// TIA Portal V19 program export: 1 tag tables, 0 data types, 19 data blocks, 18 code blocks (in call order from the OBs), 296 instance data blocks

VAR_GLOBAL   // PLC tag table "Default tag table"
   "CPU RUN" AT %I0.0 : Bool;
   "SPARE(1)" AT %I0.1 : Bool;
   "SPARE(2)" AT %I0.2 : Bool;
   "P-201 A RO 1 FEED PUMP TRIP" AT %I0.3 : Bool;
   "P-201 B RO 1 FEED PUMP TRIP" AT %I0.4 : Bool;
   "P-201 C RO 1 FEED PUMP TRIP" AT %I0.5 : Bool;
   "P-301 A RO 1 HPP PUMP TRIP" AT %I0.6 : Bool;
   "P-301 B RO B HPP PUMP TRIP" AT %I0.7 : Bool;
   "P-401 A RO 2 FEED PUMP TRIP" AT %I1.0 : Bool;
   "P-401 B RO 2 FEED PUMP TRIP" AT %I1.1 : Bool;
   "P-401 C RO 2 FEED PUMP TRIP" AT %I1.2 : Bool;
   "P 401 A RO 2 HPP PUMP TRIP" AT %I1.3 : Bool;
   "P-401 B RO 2 HPP PUMP TRIP" AT %I1.4 : Bool;
   "LPS 301 RO 1" AT %I1.5 : Bool;
   "P-202 A RO 1 FEED PUMP" AT %Q0.0 : Bool;
   "P-202 B RO 1 FEED PUMP" AT %Q0.1 : Bool;
   "P-202 C RO 1 FEED PUMP" AT %Q0.2 : Bool;
   "P-301 A RO 1 HPP PUMP" AT %Q0.3 : Bool;
   "P-301 B RO 1 HPP PUMP" AT %Q0.4 : Bool;
   "P-401 A RO 2 FEED PUMP" AT %Q0.5 : Bool;
   "P-401 B RO 2 FEED PUMP" AT %Q0.6 : Bool;
   "P-401 C RO 2 FEED PUMP" AT %Q0.7 : Bool;
   "P-402  A RO 2 HPP" AT %Q1.0 : Bool;
   "P-402 B" AT %Q1.1 : Bool;
   "HPS-301 RO 1 PRESSURE SWITCH" AT %I8.0 : Bool;
   "LPS-302 RO 1 PRESSURE SWITCH" AT %I8.1 : Bool;
   "HPS-302 RO 1 PRESSURE SWITCH" AT %I8.2 : Bool;
   "LPS-401 RO 2 PRESSURE SWITCH" AT %I8.3 : Bool;
   "HPS-401 RO 2 PRESSURE SWITCH" AT %I8.4 : Bool;
   "LPS-402 RO 2 PRESSURE SWITCH" AT %I8.5 : Bool;
   "HPS-402 RO 2 PRESSURE SWITCH" AT %I8.6 : Bool;
   "DP-703 RO 1 DOSER LEVEL SWITCH" AT %I8.7 : Bool;
   "DP-704 RO 1 DOSER LEVEL SWITCH" AT %I9.0 : Bool;
   "DP-705 RO 1 DOSER LEVEL SWITCH" AT %I9.1 : Bool;
   "P-501 A EDI FEED PUMP TRIP" AT %I9.2 : Bool;
   "P-501 B EDI FEED PUMP TRIP" AT %I9.3 : Bool;
   "P-501 C EDI FEED PUMP TRIP" AT %I9.4 : Bool;
   "EDI 501 A TRIP" AT %I9.5 : Bool;
   "EDI 501 B TRIP" AT %I9.6 : Bool;
   "P-501 A EDI FEED PUMP" AT %Q8.0 : Bool;
   "P-501 B EDI FEED PUMP" AT %Q8.1 : Bool;
   "P-501 C EDI FEED PUMP" AT %Q8.2 : Bool;
   "EDI 501" AT %Q8.3 : Bool;
   "EDI 502" AT %Q8.4 : Bool;
   "DP 703" AT %Q8.5 : Bool;
   "DP 704" AT %Q8.6 : Bool;
   "DP 705" AT %Q8.7 : Bool;
   "ABV 301" AT %Q9.0 : Bool;
   "ABV 302" AT %Q9.1 : Bool;
   "AGLV-301" AT %Q9.2 : Bool;
   "AGLV-302" AT %Q9.3 : Bool;
   "AGLV-401" AT %Q9.4 : Bool;
   "AGLV-402" AT %Q9.5 : Bool;
   "AGLV-501" AT %Q9.6 : Bool;
   "AGLV-502" AT %Q9.7 : Bool;
   "P-201 A RO 1 FEED PUMP FEED BACK" AT %I12.0 : Bool;
   "P-201 B RO 1 FEED PUMP FEED BACK" AT %I12.1 : Bool;
   "P-201 C RO 1 FEED PUMP FEED BACK" AT %I12.2 : Bool;
   "P-301 A RO 1 HPP PUMP FEED BACK" AT %I12.3 : Bool;
   "P-301 B RO 1 HPP PUMP FEED BACK" AT %I12.4 : Bool;
   "P-401 A R0 2 FEED PUMP FEED BACK" AT %I12.5 : Bool;
   "P-401 B RO 2 FEED PUMP FEED BACK" AT %I12.6 : Bool;
   "P-401 C RO 2 FEED PUMP FEED BACK" AT %I12.7 : Bool;
   "P-402 A RO 2 HPP PUMP FEED BACK" AT %I13.0 : Bool;
   "P-402 B RO 2 HPP PUMP FEED BACK" AT %I13.1 : Bool;
   "P-501 A EDI FEED PUMP FEED BACK" AT %I13.2 : Bool;
   "P-501 B EDI FEED PUMP FEED BACK" AT %I13.3 : Bool;
   "P-501 C EDI FEED PUMP FEED BACK" AT %I13.4 : Bool;
   "SPARE(3)" AT %I13.5 : Bool;
   "ABFV-301 FEED BACK OPEN" AT %I13.6 : Bool;
   "ABFV-301 FEED BACK CLOSE" AT %I13.7 : Bool;
   "ABFV-302 OPEN FEED BACK" AT %I16.0 : Bool;
   "ABFV-302 CLOSE FEED BACK" AT %I16.1 : Bool;
   "AGLV-301 OPEN FEED BACK" AT %I16.2 : Bool;
   "AGLV-301 CLOSE FEED BACK" AT %I16.3 : Bool;
   "AGLV-302 OPEN FEED BACK" AT %I16.4 : Bool;
   "AGLV-302 CLOSE FEED BACK" AT %I16.5 : Bool;
   "AGLV-401 OPEN FEED BACK" AT %I16.6 : Bool;
   "AGLV-401 CLOSE FEED BACK" AT %I16.7 : Bool;
   "AGLV-402 OPEN FEED BACK" AT %I17.0 : Bool;
   "AGLV-402 CLOSE FEED BACK" AT %I17.1 : Bool;
   "AGLV-501OPEN FEED BACK" AT %I17.2 : Bool;
   "AGLV-501 CLOSE FEED BACK" AT %I17.3 : Bool;
   "AGLV-502 OPEN FEED BACK" AT %I17.4 : Bool;
   "AGLV-502 CLOSE FEED BACK" AT %I17.5 : Bool;
   "SPARE(4)" AT %I17.6 : Bool;
   "SPARE(5)" AT %I17.7 : Bool;
   "OXIDATION REDUCTION POTENTIO METER 301" AT %IW144 : Int;
   "CONDUCTIVITY INDUCTOR CUM TRANSMITTER 301" AT %IW146 : Int;
   "PH INDICATOR CUM TRANSMITTER 301" AT %IW148 : Int;
   "PH INDICATOR CUM TRANSMITTER 302" AT %IW150 : Int;
   "CONDUCTIVITY INDICATOR CUM TRANSMITTER 302" AT %IW152 : Int;
   "LEVEL TRANSMITTER 401" AT %IW154 : Int;
   "PH INDICATOR CUM TRANSMITTER 401" AT %IW156 : Int;
   "CONDUCTIVITY INDICATOR CUM TRANSMITTER 401" AT %IW158 : Int;
   "CONFUCTIVITY INDICATOR CUM TRANSMITTER 402" AT %IW160 : Int;
   "PH INDICATOR CUM TRANSMITTER 402" AT %IW162 : Int;
   "LEVEL TRANSMITTER 501" AT %IW164 : Int;
   "FLOW INDICATOR TOTALOZER 501" AT %IW166 : Int;
   "PRESSURE TRANSMITTER 501" AT %IW168 : Int;
   "FLOW INDICATOR TRANSMITTER 502" AT %IW170 : Int;
   "PRESSURE TRANSMITTER 502" AT %IW172 : Int;
   "PRESSURE TRANSMITTER 503" AT %IW174 : Int;
   "PRESSURE TRANSMITTER 504" AT %IW176 : Int;
   "PRESSURE TRANSMITTER 505" AT %IW178 : Int;
   "PRESSURE TRANSMITTER 506" AT %IW180 : Int;
   "PH INDICATOR CUM TRANSMITTER 501" AT %IW182 : Int;
   "PH INDICATOR CUM TRANSMITTER 502" AT %IW184 : Int;
   "RESISTIVITY CUM TRANSMITTER 501" AT %IW186 : Int;
   "RESISTIVITY CUM TRANSMITTER 502" AT %IW188 : Int;
   "LEVEL TRANSMITTER 502" AT %IW190 : Int;
   "FLOW INDICATOR TRANSMITTER 503" AT %IW192 : Int;
   "FLOW INDICATOR TRANSMITTER 504" AT %IW194 : Int;
   "FLOW INDICATOR TRANSMITTER 505" AT %IW196 : Int;
   "FLOW INDICATOR TRANSMITTER 506" AT %IW198 : Int;
   "FLOW INDICATOR TRANSMITTER 507" AT %IW200 : Int;
   "FLOW INDICATOR TRANSMITTER 508" AT %IW202 : Int;
   "SPARE(6)" AT %IW204 : Int;
   "SPARE(7)" AT %IW206 : Int;
   "SPARE(8)" AT %I9.7 : Bool;
   Tag_1 AT %Q1.2 : Bool;
   Tag_2 AT %I1.6 : Bool;
   Clock_Byte AT %MB0 : Byte;
   Clock_10Hz AT %M0.0 : Bool;
   Clock_5Hz AT %M0.1 : Bool;
   "Clock_2.5Hz" AT %M0.2 : Bool;
   Clock_2Hz AT %M0.3 : Bool;
   "Clock_1.25Hz" AT %M0.4 : Bool;
   Clock_1Hz AT %M0.5 : Bool;
   "Clock_0.625Hz" AT %M0.6 : Bool;
   "Clock_0.5Hz" AT %M0.7 : Bool;
   System_Byte AT %MB1 : Byte;
   FirstScan AT %M1.0 : Bool;
   DiagStatusUpdate AT %M1.1 : Bool;
   AlwaysTRUE AT %M1.2 : Bool;
   AlwaysFALSE AT %M1.3 : Bool;
   "PLC_2 HOOTER" AT %M2.0 : Bool;
   "SET TIME" AT %MW4 : Int;
   "LT 201" AT %MD6 : Real;
   TAG122 AT %M2.1 : Bool;
   TEST_1 AT %M2.2 : Bool;
   TEST_2 AT %M2.3 : Bool;
   TEST_3 AT %M2.4 : Bool;
   GGG AT %M2.5 : Bool;
   GGG1 AT %M2.6 : Bool;
   HH AT %M2.7 : Bool;
   HOOTER AT %M3.0 : Bool;
   QQQ AT %M3.1 : Bool;
   YYU AT %M3.2 : Bool;
   YYY1 AT %M3.3 : Bool;
   YYY2 AT %M3.4 : Bool;
   SLAVE1_WRITE_DONE AT %M3.5 : Bool;
   SLAVE1_WRITE_BUSY AT %M3.6 : Bool;
   SLAVE1_WRITE_ERROR AT %M3.7 : Bool;
   CYCLE AT %MW10 : Int;
   HHH AT %M12.0 : Bool;
   Tag_3 AT %IW64 : Int;
   Tag_4 AT %IW100 : Int;
   KKKK AT %MW14 : Int;
   KKK AT %M12.1 : Bool;
   JJJJ AT %M12.2 : Bool;
   hvvvvhh AT %M12.3 : Bool;
   kkkkk AT %M12.4 : Bool;
   FFF AT %M12.5 : Bool;
   FFF1 AT %M12.6 : Bool;
END_VAR

DATA_BLOCK "DATA RECIEVED FROM MASTER DB"   // DB228
{ S7_Optimized_Access := 'FALSE' }
// stored: AutoNumber false
   VAR
      "REAL" : Real;
      REAL_1 : Real;
      REAL_2 : Real;
      REAL_3 : Real;
      REAL_4 : Real;
      REAL_5 : Real;
   END_VAR
BEGIN
END_DATA_BLOCK

DATA_BLOCK "MODBUS DB"   // DB53
{ S7_Optimized_Access := 'FALSE' }
   VAR
      "STEP" : Int;
      EDGE : Bool;
      P_TRIG : Struct
         "0" : Bool;
         "1" : Bool;
         "2" : Bool;
         "3" : Bool;
         "4" : Bool;
         "5" : Bool;
         "6" : Bool;
         "7" : Bool;
         "8" : Bool;
         "9" : Bool;
         "10" : Bool;
         "11" : Bool;
         "12" : Bool;
         "13" : Bool;
         "14" : Bool;
         "15" : Bool;
         "16" : Bool;
         "17" : Bool;
         "18" : Bool;
         "19" : Bool;
         "20" : Bool;
         "21" : Bool;
         "22" : Bool;
         "23" : Bool;
         "24" : Bool;
         "25" : Bool;
         "26" : Bool;
         "27" : Bool;
         "28" : Bool;
         "29" : Bool;
         "30" : Bool;
         "31" : Bool;
         "32" : Bool;
         "33" : Bool;
         "34" : Bool;
         "35" : Bool;
         "36" : Bool;
         "37" : Bool;
         "38" : Bool;
         "39" : Bool;
         "40" : Bool;
         "41" : Bool;
         "42" : Bool;
         "43" : Bool;
         "44" : Bool;
         "45" : Bool;
         "46" : Bool;
         "47" : Bool;
         "48" : Bool;
         "49" : Bool;
         "50" : Bool;
      END_STRUCT;
      VFD_1 : Struct
         WRITE : Struct
            DONE : Bool;
            BUSY : Bool;
            ERROR : Bool;
            STATUS : Int;
         END_STRUCT;
         READ : Struct
            DONE : Bool;
            BUSY : Bool;
            ERROR : Bool;
            STATUS : Int;
         END_STRUCT;
      END_STRUCT;
      "VFD_1 SEND" : UInt;
      "VFD_1 RECEIVE" : UInt;
      VFD_2 : Struct
         WRITE : Struct
            DONE : Bool;
            BUSY : Bool;
            ERROR : Bool;
            STATUS : Int;
         END_STRUCT;
         READ : Struct
            DONE : Bool;
            BUSY : Bool;
            ERROR : Bool;
            STATUS : Int;
         END_STRUCT;
      END_STRUCT;
      "VFD_2 SEND" : UInt;
      "VFD_2 RECEIVE" : UInt;
      VFD_3 : Struct
         WRITE : Struct
            DONE : Bool;
            BUSY : Bool;
            ERROR : Bool;
            STATUS : Int;
         END_STRUCT;
         READ : Struct
            DONE : Bool;
            BUSY : Bool;
            ERROR : Bool;
            STATUS : Int;
         END_STRUCT;
      END_STRUCT;
      "VFD_3 SEND" : UInt;
      "VFD_3 RECEIVE" : UInt;
      VFD_4 : Struct
         WRITE : Struct
            DONE : Bool;
            BUSY : Bool;
            ERROR : Bool;
            STATUS : Int;
         END_STRUCT;
         READ : Struct
            DONE : Bool;
            BUSY : Bool;
            ERROR : Bool;
            STATUS : Int;
         END_STRUCT;
      END_STRUCT;
      "VFD_4 SEND" : UInt;
      "VFD_4 RECEIVE" : UInt;
      VFD_5 : Struct
         WRITE : Struct
            DONE : Bool;
            BUSY : Bool;
            ERROR : Bool;
            STATUS : Int;
         END_STRUCT;
         READ : Struct
            DONE : Bool;
            BUSY : Bool;
            ERROR : Bool;
            STATUS : Int;
         END_STRUCT;
      END_STRUCT;
      "VFD_5 SEND" : UInt;
      "VFD_5 RECEIVE" : UInt;
      VFD_6 : Struct
         WRITE : Struct
            DONE : Bool;
            BUSY : Bool;
            ERROR : Bool;
            STATUS : Int;
         END_STRUCT;
         READ : Struct
            DONE : Bool;
            BUSY : Bool;
            ERROR : Bool;
            STATUS : Int;
         END_STRUCT;
      END_STRUCT;
      "VFD_6 SEND" : UInt;
      "VFD_6 RECEIVE" : UInt;
      VFD_7 : Struct
         WRITE : Struct
            DONE : Bool;
            BUSY : Bool;
            ERROR : Bool;
            STATUS : Int;
         END_STRUCT;
         READ : Struct
            DONE : Bool;
            BUSY : Bool;
            ERROR : Bool;
            STATUS : Int;
         END_STRUCT;
      END_STRUCT;
      "VFD_7 SEND" : UInt;
      "VFD_7 RECEIVE" : UInt;
   END_VAR
BEGIN
END_DATA_BLOCK

DATA_BLOCK "AI SCALING DB"   // DB5
{ S7_Optimized_Access := 'FALSE' }
   VAR RETAIN
      SET : Struct
         "OXIDATION REDUCTION POTENTIO METER 301" : Int;
         "CONDUCTIVITY INDUCTOR CUM TRANSMITTER 301" : Int;
         "PH INDICATOR CUM TRANSMITTER 301" : Int;
         "PH INDICATOR CUM TRANSMITTER 302" : Int;
         "CONDUCTIVITY INDICATOR CUM TRANSMITTER 302" : Int;
         "LEVEL TRANSMITTER 401" : Int;
         "PH INDICATOR CUM TRANSMITTER 401" : Int;
         "CONDUCTIVITY INDICATOR CUM TRANSMITTER 401" : Int;
         "CONFUCTIVITY INDICATOR CUM TRANSMITTER 402" : Int;
         "PH INDICATOR CUM TRANSMITTER 402" : Int;
         "LEVEL TRANSMITTER 501" : Int;
         "FLOW INDICATOR TOTALOZER 501" : Int;
         "PRESSURE TRANSMITTER 501" : Int;
         "FLOW INDICATOR TRANSMITTER 502" : Int;
         "PRESSURE TRANSMITTER 502" : Int;
         "PRESSURE TRANSMITTER 503" : Int;
         "PRESSURE TRANSMITTER 504" : Int;
         "PRESSURE TRANSMITTER 505" : Int;
         "PRESSURE TRANSMITTER 506" : Int;
         "PH INDICATOR CUM TRANSMITTER 501" : Int;
         "PH INDICATOR CUM TRANSMITTER 502" : Int;
         "RESISTIVITY CUM TRANSMITTER 501" : Int;
         "RESISTIVITY CUM TRANSMITTER 502" : Int;
         "LEVEL TRANSMITTER 502" : Int;
         "FLOW INDICATOR TRANSMITTER 503" : Int;
         "FLOW INDICATOR TRANSMITTER 504" : Int;
         "FLOW INDICATOR TRANSMITTER 505" : Int;
         "FLOW INDICATOR TRANSMITTER 506" : Int;
         "FLOW INDICATOR TRANSMITTER 507" : Int;
         "FLOW INDICATOR TRANSMITTER 508" : Int;
         "SPARE(6)" : Int;
         "SPARE(7)" : Int;
      END_STRUCT;
      MIN : Struct
         "OXIDATION REDUCTION POTENTIO METER 301" { S7_SetPoint := 'True'} : Real := -1900.0;
         "CONDUCTIVITY INDUCTOR CUM TRANSMITTER 301" { S7_SetPoint := 'True'} : Real;
         "PH INDICATOR CUM TRANSMITTER 301" { S7_SetPoint := 'True'} : Real;
         "PH INDICATOR CUM TRANSMITTER 302" { S7_SetPoint := 'True'} : Real;
         "CONDUCTIVITY INDICATOR CUM TRANSMITTER 302" { S7_SetPoint := 'True'} : Real;
         "LEVEL TRANSMITTER 401" { S7_SetPoint := 'True'} : Real;
         "PH INDICATOR CUM TRANSMITTER 401" { S7_SetPoint := 'True'} : Real;
         "CONDUCTIVITY INDICATOR CUM TRANSMITTER 401" { S7_SetPoint := 'True'} : Real;
         "CONFUCTIVITY INDICATOR CUM TRANSMITTER 402" { S7_SetPoint := 'True'} : Real;
         "PH INDICATOR CUM TRANSMITTER 402" { S7_SetPoint := 'True'} : Real;
         "LEVEL TRANSMITTER 501" { S7_SetPoint := 'True'} : Real;
         "FLOW INDICATOR TOTALOZER 501" { S7_SetPoint := 'True'} : Real;
         "PRESSURE TRANSMITTER 501" { S7_SetPoint := 'True'} : Real;
         "FLOW INDICATOR TRANSMITTER 502" { S7_SetPoint := 'True'} : Real;
         "PRESSURE TRANSMITTER 502" : Real;
         "PRESSURE TRANSMITTER 503" : Real;
         "PRESSURE TRANSMITTER 504" : Real;
         "PRESSURE TRANSMITTER 505" : Real;
         "PRESSURE TRANSMITTER 506" : Real;
         "PH INDICATOR CUM TRANSMITTER 501" : Real;
         "PH INDICATOR CUM TRANSMITTER 502" : Real;
         "RESISTIVITY CUM TRANSMITTER 501" : Real;
         "RESISTIVITY CUM TRANSMITTER 502" : Real;
         "LEVEL TRANSMITTER 502" : Real;
         "FLOW INDICATOR TRANSMITTER 503" : Real;
         "FLOW INDICATOR TRANSMITTER 504" : Real;
         "FLOW INDICATOR TRANSMITTER 505" : Real;
         "FLOW INDICATOR TRANSMITTER 506" : Real;
         "FLOW INDICATOR TRANSMITTER 507" : Real;
         "FLOW INDICATOR TRANSMITTER 508" : Real;
         "SPARE(6)" : Real;
         "SPARE(7)" : Real;
      END_STRUCT;
      MAX : Struct
         "OXIDATION REDUCTION POTENTIO METER 301" { S7_SetPoint := 'True'} : Real := 1900.0;
         "CONDUCTIVITY INDUCTOR CUM TRANSMITTER 301" { S7_SetPoint := 'True'} : Real := 1999.0;
         "PH INDICATOR CUM TRANSMITTER 301" { S7_SetPoint := 'True'} : Real := 14.0;
         "PH INDICATOR CUM TRANSMITTER 302" { S7_SetPoint := 'True'} : Real := 14.0;
         "CONDUCTIVITY INDICATOR CUM TRANSMITTER 302" { S7_SetPoint := 'True'} : Real := 1999.0;
         "LEVEL TRANSMITTER 401" { S7_SetPoint := 'True'} : Real := 100.0;
         "PH INDICATOR CUM TRANSMITTER 401" { S7_SetPoint := 'True'} : Real := 14.0;
         "CONDUCTIVITY INDICATOR CUM TRANSMITTER 401" { S7_SetPoint := 'True'} : Real := 1999.0;
         "CONFUCTIVITY INDICATOR CUM TRANSMITTER 402" { S7_SetPoint := 'True'} : Real := 1999.0;
         "PH INDICATOR CUM TRANSMITTER 402" { S7_SetPoint := 'True'} : Real := 14.0;
         "LEVEL TRANSMITTER 501" { S7_SetPoint := 'True'} : Real := 100.0;
         "FLOW INDICATOR TOTALOZER 501" { S7_SetPoint := 'True'} : Real := 14.0;
         "PRESSURE TRANSMITTER 501" { S7_SetPoint := 'True'} : Real := 6.0;
         "FLOW INDICATOR TRANSMITTER 502" { S7_SetPoint := 'True'} : Real := 14.0;
         "PRESSURE TRANSMITTER 502" { S7_SetPoint := 'True'} : Real := 6.0;
         "PRESSURE TRANSMITTER 503" { S7_SetPoint := 'True'} : Real := 6.0;
         "PRESSURE TRANSMITTER 504" { S7_SetPoint := 'True'} : Real := 6.0;
         "PRESSURE TRANSMITTER 505" { S7_SetPoint := 'True'} : Real := 6.0;
         "PRESSURE TRANSMITTER 506" { S7_SetPoint := 'True'} : Real := 6.0;
         "PH INDICATOR CUM TRANSMITTER 501" { S7_SetPoint := 'True'} : Real := 14.0;
         "PH INDICATOR CUM TRANSMITTER 502" { S7_SetPoint := 'True'} : Real := 14.0;
         "RESISTIVITY CUM TRANSMITTER 501" { S7_SetPoint := 'True'} : Real := 100.0;
         "RESISTIVITY CUM TRANSMITTER 502" { S7_SetPoint := 'True'} : Real := 100.0;
         "LEVEL TRANSMITTER 502" { S7_SetPoint := 'True'} : Real := 100.0;
         "FLOW INDICATOR TRANSMITTER 503" { S7_SetPoint := 'True'} : Real := 5.0;
         "FLOW INDICATOR TRANSMITTER 504" { S7_SetPoint := 'True'} : Real := 5.0;
         "FLOW INDICATOR TRANSMITTER 505" { S7_SetPoint := 'True'} : Real := 1000.0;
         "FLOW INDICATOR TRANSMITTER 506" { S7_SetPoint := 'True'} : Real := 150.0;
         "FLOW INDICATOR TRANSMITTER 507" { S7_SetPoint := 'True'} : Real := 150.0;
         "FLOW INDICATOR TRANSMITTER 508" { S7_SetPoint := 'True'} : Real := 1000.0;
         "SPARE(6)" { S7_SetPoint := 'True'} : Real;
         "SPARE(7)" : Real;
      END_STRUCT;
      PV : Struct
         "OXIDATION REDUCTION POTENTIO METER 301" : Real;
         "CONDUCTIVITY INDUCTOR CUM TRANSMITTER 301" : Real;
         "PH INDICATOR CUM TRANSMITTER 301" : Real;
         "PH INDICATOR CUM TRANSMITTER 302" : Real;
         "CONDUCTIVITY INDICATOR CUM TRANSMITTER 302" : Real;
         "LEVEL TRANSMITTER 401" : Real;
         "PH INDICATOR CUM TRANSMITTER 401" : Real;
         "CONDUCTIVITY INDICATOR CUM TRANSMITTER 401" : Real;
         "CONFUCTIVITY INDICATOR CUM TRANSMITTER 402" : Real;
         "PH INDICATOR CUM TRANSMITTER 402" : Real;
         "LEVEL TRANSMITTER 501" : Real;
         "FLOW INDICATOR TOTALOZER 501" : Real;
         "PRESSURE TRANSMITTER 501" : Real;
         "FLOW INDICATOR TRANSMITTER 502" : Real;
         "PRESSURE TRANSMITTER 502" : Real;
         "PRESSURE TRANSMITTER 503" : Real;
         "PRESSURE TRANSMITTER 504" : Real;
         "PRESSURE TRANSMITTER 505" : Real;
         "PRESSURE TRANSMITTER 506" : Real;
         "PH INDICATOR CUM TRANSMITTER 501" : Real;
         "PH INDICATOR CUM TRANSMITTER 502" : Real;
         "RESISTIVITY CUM TRANSMITTER 501" : Real;
         "RESISTIVITY CUM TRANSMITTER 502" : Real;
         "LEVEL TRANSMITTER 502" : Real;
         "FLOW INDICATOR TRANSMITTER 503" : Real;
         "FLOW INDICATOR TRANSMITTER 504" : Real;
         "FLOW INDICATOR TRANSMITTER 505" : Real;
         "FLOW INDICATOR TRANSMITTER 506" : Real;
         "FLOW INDICATOR TRANSMITTER 507" : Real;
         "FLOW INDICATOR TRANSMITTER 508" : Real;
         "SPARE(6)" : Real;
         "SPARE(7)" : Real;
      END_STRUCT;
      SPARE : Bool;
      SPARE_1 : Bool;
      "LT-401" : Struct
         LOW_BUFF : Int;
         HIGH_BUFF : Int;
      END_STRUCT;
      "LT-501" : Struct
         LOW_BUFF : Int;
         HIGH_BUFF : Int;
      END_STRUCT;
      "LT-502" : Struct
         LOW_BUFF : Int;
         HIGH_BUFF : Int;
      END_STRUCT;
      "LT-401 SET VALVE" : Struct
         LL : Real;
         L : Real;
         H : Real;
         HH : Real;
      END_STRUCT;
      "LT-501 SET VALVE" : Struct
         LL : Real;
         L : Real;
         H : Real;
         HH : Real;
      END_STRUCT;
      "LT-502 SET VALVE" : Struct
         LL : Real;
         L : Real;
         H : Real;
         HH : Real;
      END_STRUCT;
   END_VAR
BEGIN
END_DATA_BLOCK

DATA_BLOCK "AO SCALING DB"   // DB170
{ S7_Optimized_Access := 'FALSE' }
   VAR
      SET : Struct
         "VFD P-301A" : Real;
         "VFD P-301B" : Real;
         "VFD P-402A" : Real;
         "VFD P-402B" : Real;
      END_STRUCT;
      MIN : Struct
         "VFD P-301A" : Real;
         "VFD P-301B" : Real;
         "VFD P-402A" : Real;
         "VFD P-402B" : Real;
         "VFD P-501A_7" : Real;
      END_STRUCT;
      MAX : Struct
         "VFD P-301A" { S7_SetPoint := 'True'} : Real := 50.0;
         "VFD P-301B" { S7_SetPoint := 'True'} : Real := 50.0;
         "VFD P-402A" { S7_SetPoint := 'True'} : Real := 50.0;
         "VFD P-402B" { S7_SetPoint := 'True'} : Real := 50.0;
         "VFD P-501A_7" : Real;
      END_STRUCT;
      PV : Struct
         "VFD P-301A" : Int;
         "VFD P-301B" : Int;
         "VFD P-402A" : Int;
         "VFD P-402B" : Int;
      END_STRUCT;
   END_VAR
BEGIN
END_DATA_BLOCK

DATA_BLOCK "FLUSHING VAVLE DB"   // DB63
{ S7_Optimized_Access := 'TRUE' }
// stored: MemoryReserve 100
   VAR
      "ABV 301" : Bool;
      "ABV 302" : Bool;
      "AGLV-301" : Bool;
      "AGLV-302" : Bool;
      "AGLV-401" : Bool;
      "AGLV-402" : Bool;
      "ABFV 501" : Bool;
      "ABFV 502" : Bool;
      "ABV 301 CLOSE VALVE" : Bool;
      "ABV 302 CLOSE VALVE" : Bool;
      "AGLV 301 CLOSE VALVE" : Bool;
      "AGLV 302 CLOSE VALVE" : Bool;
      "AGLV 401 CLOSE VALVE" : Bool;
      "AGLV-402 CLOSE VALVE" : Bool;
      "ABFV 501 CLOSE VALVE" : Bool;
      "ABFV 502 CLOSE VALVE" : Bool;
   END_VAR
BEGIN
END_DATA_BLOCK

DATA_BLOCK "INPUT MAPING DB"   // DB1
{ S7_Optimized_Access := 'FALSE' }
   VAR
      "CIP RUN" : Bool;
      "SPARE(1)" : Bool;
      "SPARE(2)" : Bool;
      "P-201 A RO 1 FEED PUMP TRIP" : Bool;
      "P-201 B RO 1 FEED PUMP TRIP" : Bool;
      "P-201 C RO 1 FEED PUMP TRIP" : Bool;
      "P-301 A RO 1 HPP PUMP TRIP" : Bool;
      "P-301 B RO B HPP PUMP TRIP" : Bool;
      "P-401 A RO 2 FEED PUMP TRIP" : Bool;
      "P-401 B RO 2 FEED PUMP TRIP" : Bool;
      "P-401 C RO 2 FEED PUMP TRIP" : Bool;
      "P 401 A RO 2 HPP PUMP TRIP" : Bool;
      "P-401 B RO 2 HPP PUMP TRIP" : Bool;
      "LPS 301 RO 1" : Bool;
      "HPS-301 RO 1 PRESSURE SWITCH" : Bool;
      "LPS-302 RO 1 PRESSURE SWITCH" : Bool;
      "HPS-302 RO 1 PRESSURE SWITCH" : Bool;
      "LPS-401 RO 2 PRESSURE SWITCH" : Bool;
      "HPS-401 RO 2 PRESSURE SWITCH" : Bool;
      "LPS-402 RO 2 PRESSURE SWITCH" : Bool;
      "HPS-402 RO 2 PRESSURE SWITCH" : Bool;
      "DP-703 RO 1 DOSER LEVEL SWITCH" : Bool;
      "DP-704 RO 1 DOSER LEVEL SWITCH" : Bool;
      "DP-705 RO 1 DOSER LEVEL SWITCH" : Bool;
      "P-501 A EDI FEED PUMP TRIP" : Bool;
      "P-501 B EDI FEED PUMP TRIP" : Bool;
      "P-501 C EDI FEED PUMP TRIP" : Bool;
      "EDI 501 A TRIP" : Bool;
      "EDI 501 B TRIP" : Bool;
      "SPARE(8)" : Bool;
      "P-201 A RO 1 FEED PUMP FEED BACK" : Bool;
      "P-201 B RO 1 FEED PUMP FEED BACK" : Bool;
      "P-201 C RO 1 FEED PUMP FEED BACK" : Bool;
      "P-301 A RO 1 HPP PUMP FEED BACK" : Bool;
      "P-301 B RO 1 HPP PUMP FEED BACK" : Bool;
      "P-401 A R0 2 FEED PUMP FEED BACK" : Bool;
      "P-401 B RO 2 FEED PUMP FEED BACK" : Bool;
      "P-401 C RO 2 FEED PUMP FEED BACK" : Bool;
      "P-402 A RO 2 HPP PUMP FEED BACK" : Bool;
      "P-402 B RO 2 HPP PUMP FEED BACK" : Bool;
      "P-501 A EDI FEED PUMP FEED BACK" : Bool;
      "P-501 B EDI FEED PUMP FEED BACK" : Bool;
      "P-501 C EDI FEED PUMP FEED BACK" : Bool;
      "SPARE(3)" : Bool;
      "ABFV-301 FEED BACK OPEN" : Bool;
      "ABFV-301 FEED BACK CLOSE" : Bool;
      "ABFV-302 OPEN FEED BACK" : Bool;
      "ABFV-302 CLOSE FEED BACK" : Bool;
      "AGLV-301 OPEN FEED BACK" : Bool;
      "AGLV-301 CLOSE FEED BACK" : Bool;
      "AGLV-302 OPEN FEED BACK" : Bool;
      "AGLV-302 CLOSE FEED BACK" : Bool;
      "AGLV-401 OPEN FEED BACK" : Bool;
      "AGLV-401 CLOSE FEED BACK" : Bool;
      "AGLV-402 OPEN FEED BACK" : Bool;
      "AGLV-402 CLOSE FEED BACK" : Bool;
      "AGLV-501OPEN FEED BACK" : Bool;
      "AGLV-501 CLOSE FEED BACK" : Bool;
      "AGLV-502 OPEN FEED BACK" : Bool;
      "AGLV-502 CLOSE FEED BACK" : Bool;
      "SPARE(4)" : Bool;
      "SPARE(5)" : Bool;
   END_VAR
BEGIN
END_DATA_BLOCK

DATA_BLOCK "OUTPUT MAPING DB PLC 2"   // DB2
{ S7_Optimized_Access := 'FALSE' }
   VAR
      "P-202 A RO 1 FEED PUMP" : Bool;
      "P-202 B RO 1 FEED PUMP" : Bool;
      "P-202 C RO 1 FEED PUMP" : Bool;
      "P-301 A RO 1 HPP PUMP" : Bool;
      "P-301 B RO 1 HPP PUMP" : Bool;
      "P-401 A RO 2 FEED PUMP" : Bool;
      "P-401 B RO 2 FEED PUMP" : Bool;
      "P-401 C RO 2 FEED PUMP" : Bool;
      "P-402  A RO 2 HPP" : Bool;
      "P-402 B" : Bool;
      "P-501 A EDI FEED PUMP" : Bool;
      "P-501 B EDI FEED PUMP" : Bool;
      "P-501 C EDI FEED PUMP" : Bool;
      "EDI 501" : Bool;
      "EDI 502" : Bool;
      "DP 703" : Bool;
      "DP 704" : Bool;
      "DP 705" : Bool;
      "ABV 301" : Bool;
      "ABV 302" : Bool;
      "AGLV-301" : Bool;
      "AGLV-302" : Bool;
      "AGLV-401" : Bool;
      "AGLV-402" : Bool;
      "AGLV-501" : Bool;
      "AGLV-502" : Bool;
      "HOOTER RESET" : Bool;
   END_VAR
BEGIN
END_DATA_BLOCK

DATA_BLOCK "AUTO_SUBOUTPUT DB"   // DB71
{ S7_Optimized_Access := 'TRUE' }
// stored: MemoryReserve 100
   VAR
      "P-202 A RO 1 FEED PUMP" : Bool;
      "P-202 B RO 1 FEED PUMP" : Bool;
      "P-202 C RO 1 FEED PUMP" : Bool;
      "P-301 A RO 1 HPP PUMP" : Bool;
      "P-301 B RO 1 HPP PUMP" : Bool;
      "P-401 A RO 2 FEED PUMP" : Bool;
      "P-401 B RO 2 FEED PUMP" : Bool;
      "P-401 C RO 2 FEED PUMP" : Bool;
      "P-402  A RO 2 HPP" : Bool;
      "P-402 B" : Bool;
      "P-501 A EDI FEED PUMP" : Bool;
      "P-501 B EDI FEED PUMP" : Bool;
      "P-501 C EDI FEED PUMP" : Bool;
      "EDI 501" : Bool;
      "EDI 502" : Bool;
      "DP 703" : Bool;
      "DP 704" : Bool;
      "DP 705" : Bool;
      "ABV 301" : Bool;
      "ABV 302" : Bool;
      "AGLV-301" : Bool;
      "AGLV-302" : Bool;
      "AGLV-401" : Bool;
      "AGLV-402" : Bool;
      "AGLV-501" : Bool;
      "AGLV-502" : Bool;
   END_VAR
BEGIN
END_DATA_BLOCK

DATA_BLOCK "MANUAL BIT"   // DB4
{ S7_Optimized_Access := 'FALSE' }
   VAR
      "P-202 A RO 1 FEED PUMP" : Bool;
      "P-202 B RO 1 FEED PUMP" : Bool;
      "P-202 C RO 1 FEED PUMP" : Bool;
      "P-301 A RO 1 HPP PUMP" : Bool;
      "P-301 B RO 1 HPP PUMP" : Bool;
      "P-401 A RO 2 FEED PUMP" : Bool;
      "P-401 B RO 2 FEED PUMP" : Bool;
      "P-401 C RO 2 FEED PUMP" : Bool;
      "P-402  A RO 2 HPP" : Bool;
      "P-402 B" : Bool;
      "P-501 A EDI FEED PUMP" : Bool;
      "P-501 B EDI FEED PUMP" : Bool;
      "P-501 C EDI FEED PUMP" : Bool;
      "EDI 501" : Bool;
      "EDI 502" : Bool;
      "DP 703" : Bool;
      "DP 704" : Bool;
      "DP 705" : Bool;
      "ABV 301" : Bool;
      "ABV 302" : Bool;
      "AGLV-301" : Bool;
      "AGLV-302" : Bool;
      "AGLV-401" : Bool;
      "AGLV-402" : Bool;
      "AGLV-501" : Bool;
      "AGLV-502" : Bool;
      "SPARE 13" : Bool;
      "SPARE 16" : Bool;
      "SPARE 17" : Bool;
      "SPARE 18" : Bool;
      "SPARE 19" : Bool;
      "SPARE 20" : Bool;
      "SPARE 21" : Bool;
      "SPARE 22" : Bool;
      "SPARE 23" : Bool;
      "SPARE 24" : Bool;
      "SPARE 25" : Bool;
      "SPARE 26" : Bool;
      "SPARE 27" : Bool;
      "SPARE 28" : Bool;
      "SPARE 29" : Bool;
      "SPARE 30" : Bool;
   END_VAR
BEGIN
END_DATA_BLOCK

DATA_BLOCK "MODE SELECTION DB"   // DB3
{ S7_Optimized_Access := 'FALSE' }
   VAR
      "RO-1" : Struct
         AUTO : Bool;
         MANUAL : Bool;
         STANDBY : Bool;
         "MODE BUFF" : Int;
         "PROCESS BUFF" : Int;
         START : Bool;
         STOP : Bool;
      END_STRUCT;
      "RO-2" : Struct
         AUTO : Bool;
         MANUAL : Bool;
         STANDBY : Bool;
         "MODE BUFF" : Int;
         "PROCESS BUFF" : Int;
         START : Bool;
         STOP : Bool;
      END_STRUCT;
      EDI : Struct
         AUTO : Bool;
         MANUAL : Bool;
         STANDBY : Bool;
         "MODE BUFF" : Int;
         "PROCESS BUFF" : Int;
         START : Bool;
         STOP : Bool;
      END_STRUCT;
   END_VAR
BEGIN
END_DATA_BLOCK

DATA_BLOCK "PUMP SELECTION"   // DB36
{ S7_Optimized_Access := 'FALSE' }
   VAR RETAIN
      "P-202 A RO 1 FEED PUMP" : Bool;
      "P-202 B RO 1 FEED PUMP" : Bool;
      "P-202 C RO 1 FEED PUMP" : Bool;
      "P-301 RO 1 HPP PUMP A" : Bool;
      "P-301 RO 1 HPP PUMP B" : Bool;
      "P-401 A RO 2 FEED PUMP" : Bool;
      "P-401 B RO 2 FEED PUMP" : Bool;
      "P-401 C RO 2 FEED PUMP" : Bool;
      "P-402 RO 2 HPP A" : Bool;
      "P-402 RO 2 HPP B" : Bool;
      "P-501 A EDI FEED PUMP" : Bool;
      "P-501 B EDI FEED PUMP" : Bool;
      "P-501 C EDI FEED PUMP" : Bool;
      "EDI-501" : Bool;
      "EDI-502" : Bool;
   END_VAR
BEGIN
END_DATA_BLOCK

DATA_BLOCK "ALARM DB PLC 2"   // DB37
{ S7_Optimized_Access := 'FALSE' }
   VAR
      "P-201 A RO 1 FEED PUMP TRIP" : Bool;
      "P-201 B RO 1 FEED PUMP TRIP" : Bool;
      "P-201 C RO 1 FEED PUMP TRIP" : Bool;
      "P-301 A RO 1 HPP PUMP TRIP" : Bool;
      "P-301 B RO B HPP PUMP TRIP" : Bool;
      "P-401 A RO 2 FEED PUMP TRIP" : Bool;
      "P-401 B RO 2 FEED PUMP TRIP" : Bool;
      "P-401 C RO 2 FEED PUMP TRIP" : Bool;
      "P 401 A RO 2 HPP PUMP TRIP" : Bool;
      "P-401 B RO 2 HPP PUMP TRIP" : Bool;
      "P-501 A EDI FEED PUMP TRIP" : Bool;
      "P-501 B EDI FEED PUMP TRIP" : Bool;
      "P-501 C EDI FEED PUMP TRIP" : Bool;
      "EDI 501 A TRIP" : Bool;
      "EDI 501 B TRIP" : Bool;
      "P-201 A RO 1 FEED PUMP_FEEDBACK FAIL" : Bool;
      "P-201 B RO 1 FEED PUMP_FEEDBACK FAIL" : Bool;
      "P-201 C RO 1 FEED PUMP_FEEDBACK FAIL" : Bool;
      "P-301 A RO 1 HPP PUMP_FEEDBACK FAIL" : Bool;
      "P-301 B RO B HPP PUMP_FEEDBACK FAIL" : Bool;
      "P-401 A RO 2 FEED PUMP_FEEDBACK FAIL" : Bool;
      "P-401 B RO 2 FEED PUMP_FEEDBACK FAIL" : Bool;
      "P-401 C RO 2 FEED PUMP_FEEDBACK FAIL" : Bool;
      "P 401 A RO 2 HPP PUMP_FEEDBACK FAIL" : Bool;
      "P-401 B RO 2 HPP PUMP_FEEDBACK FAIL" : Bool;
      "P-501 A EDI FEED PUMP_FEEDBACK FAIL" : Bool;
      "P-501 B EDI FEED PUMP_FEEDBACK FAIL" : Bool;
      "P-501 C EDI FEED PUMP_FEEDBACK FAIL" : Bool;
      "EDI 501 A _FEEDBACK FAIL" : Bool;
      "EDI 501 B_FEEDBACK FAIL" : Bool;
      "RO-01 ORP DUMP VALVE ABV-301 OPEN COMMOND FAIL" : Bool;
      "RO-01 ORP DUMP VALVE ABV-301 CLOSE COMMOND FAIL" : Bool;
      "RO-01 ORP PROCESS VALVE ABV-302 OPEN COMMOND FAIL" : Bool;
      "RO-01 ORP PROCESS VALVE ABV-302 CLOSE COMMOND FAIL" : Bool;
      "RO-1 A AUTO FLUSING VALVE AGLV-301 OPEN COMMOND FAIL" : Bool;
      "RO-1 A AUTO FLUSING VALVE AGLV-301 CLOSE COMMOND FAIL" : Bool;
      "RO-1 B AUTO FLUSING VALVE AGLV-302 OPEN COMMOND FAIL" : Bool;
      "RO-1 B AUTO FLUSING VALVE AGLV-302 CLOSE COMMOND FAIL" : Bool;
      "RO-2 A AUTO FLUSING VALVE AGLV-401 OPEN COMMOND FAIL" : Bool;
      "RO-2 A AUTO FLUSING VALVE AGLV-401 CLOSE COMMOND FAIL" : Bool;
      "RO-2 B AUTO FLUSING VALVE AGLV-402 OPEN COMMOND FAIL" : Bool;
      "RO-2 B AUTO FLUSING VALVE AGLV-402 CLOSE COMMOND FAIL" : Bool;
      "EDI AUTO DUMP VALVE ABV-501 OPEN COMMOND FAIL" : Bool;
      "EDI AUTO DUMP VALVE ABV-501 CLOSE COMMOND FAIL" : Bool;
      "DM TANK INLET VALVE ABV-502 OPEN COMMOND FAIL" : Bool;
      "DM TANK INLET VALVE ABV-502 CLOSE COMMOND FAIL" : Bool;
      "RO-02 FEED TANK LEVEL ( LT-401)- LOW LOW" : Bool;
      "RO-02 FEED TANK LEVEL ( LT-401)- HIGH HIGH" : Bool;
      "EDI FEED TANK LEVEL ( LT-501)- LOW LOW" : Bool;
      "EDI FEED TANK LEVEL ( LT-501)- HIGH HIGH" : Bool;
      "DM WATER STORAGE TANK  LEVEL ( LT-502)- LOW LOW" : Bool;
      "DM WATER STORAGE TANK LEVEL ( LT-502)- HIGH HIGH" : Bool;
      "RO-01A LPS-301 LOW" : Bool;
      "RO-01 B LPS-302 LOW" : Bool;
      "RO-01 A HPS-301 HIGH" : Bool;
      "RO-01B HPS-302 HIGH" : Bool;
      "RO-02A LPS-401 LOW" : Bool;
      "RO-02B LPS-402 LOW" : Bool;
      "RO-02A HPS-401 HIGH" : Bool;
      "RO-02 B HPS-402 HIGH" : Bool;
      "EDI-501A FEED PRESSURE PT-501 LOW" : Bool;
      "PT-501A LOW_SET VALIDATION TIME OVER_(SYSTEM STOP)" : Bool;
      "EDI-501A FEED PRESSURE PT-501 HIGH" : Bool;
      "PT-501A HIGH_SET VALIDATION TIME OVER_(SYSTEM STOP)" : Bool;
      "EDI-501B FEED PRESSURE PT-502 LOW" : Bool;
      "PT-501B LOW_SET VALIDATION TIME OVER_(SYSTEM STOP)" : Bool;
      "EDI-501B FEED PRESSURE PT-502 HIGH" : Bool;
      "PT-501B HIGH_SET VALIDATION TIME OVER_(SYSTEM STOP)" : Bool;
      "EDI-501B CONCENTRATE OUT PRESSURE PT-503 HIGH" : Bool;
      "PT-503 HIGH_SET VALIDATION TIME OVER_(SYSTEM STOP)" : Bool;
      "EDI-501A PRODUCT OUT PRESSURE PT-504 HIGH" : Bool;
      "PT-504 HIGH_SET VALIDATION TIME OVER_(SYSTEM STOP)" : Bool;
      "EDI-501A CONCENTRATE OUT PRESSURE PT-505 HIGH" : Bool;
      "PT-505 HIGH_SET VALIDATION TIME OVER_(SYSTEM STOP)" : Bool;
      "EDI-501B PRODUCT OUT PRESSURE PT-506 HIGH" : Bool;
      "PT-506 HIGH_SET VALIDATION TIME OVER_(SYSTEM STOP)" : Bool;
      "RO-01 FEED PHIT-301 HIGH" : Bool;
      "RO-01 FEED PHIT-301 LOW" : Bool;
      "RO-01 PRODUCT PHIT-302 HIGH" : Bool;
      "RO-01 PRODUCT PHIT-302 LOW" : Bool;
      "RO-02 FEED PHIT-401 HIGH" : Bool;
      "RO-02 FEED PHIT-401 LOW" : Bool;
      "RO-02 PRODUCT PHIT-402 HIGH" : Bool;
      "RO-02 PRODUCT PHIT-402 LOW" : Bool;
      "EDI-501A PRODUCT OUT  PHIT-501 HIGH" : Bool;
      "EDI-501A PRODUCT OUT  PHIT-501 LOW" : Bool;
      "EDI-501B PRODUCT OUT  PHIT-502 HIGH" : Bool;
      "EDI-501B PRODUCT OUT PHIT-502 LOW" : Bool;
      "RO-01 FEED CIT-301 HIGH" : Bool;
      "CIT-301 HIGH_SET VALIDATION TIME OVER_(SYSTEM STOP)" : Bool;
      "RO-01 PRODUCT CIT-302 HIGH" : Bool;
      "CIT-302 HIGH_SET VALIDATION TIME OVER_(SYSTEM STOP)" : Bool;
      "RO-02 FEED CIT-401 HIGH" : Bool;
      "CIT-401 HIGH_SET VALIDATION TIME OVER_(SYSTEM STOP)" : Bool;
      "RO-02 PRODUCT CIT-402 HIGH" : Bool;
      "CIT-402 HIGH_SET VALIDATION TIME OVER_(SYSTEM STOP)" : Bool;
      "EDI-501A PRODUCT OUT RIT-501 HIGH" : Bool;
      "RIT-501A HIGH_SET VALIDATION TIME OVER_(SYSTEM STOP)" : Bool;
      "EDI-501B PRODUCT OUT RIT-502 HIGH" : Bool;
      "RIT-501B HIGH_SET VALIDATION TIME OVER_(SYSTEM STOP)" : Bool;
      "ORP-301 HIGH" : Bool;
      "ORP-301 HIGH_SET VALIDATION TIME OVER_(SYSTEM STOP)" : Bool;
      "EDI-501A FEED PRESSURE FIT-501 LOW" : Bool;
      "FIT-501  LOW_SET VALIDATION TIME OVER_(SYSTEM STOP)" : Bool;
      "EDI-501B FEED PRESSURE FIT-502 LOW" : Bool;
      "FIT-501 LOW_SET VALIDATION TIME OVER_(SYSTEM STOP)" : Bool;
      "EDI-501B CONCENTRATE OUT PRESSURE FIT-503 LOW" : Bool;
      "FIT-503 LOW_SET VALIDATION TIME OVER_(SYSTEM STOP)" : Bool;
      "EDI-501A PRODUCT OUT PRESSURE FIT-504 LOW" : Bool;
      "FIT-504 LOW_SET VALIDATION TIME OVER_(SYSTEM STOP)" : Bool;
      "EDI-501B CONCENTRATE OUT PRESSURE FIT-505 LOW" : Bool;
      "FIT-505 LOW_SET VALIDATION TIME OVER_(SYSTEM STOP)" : Bool;
      "EDI-501B CONCENTRATE OUT PRESSURE FIT-505 HIGH" : Bool;
      "FIT-505 HIGH_SET VALIDATION TIME OVER_(SYSTEM STOP)" : Bool;
      "EDI-501A PRODUCT OUT PRESSURE FIT-506 LOW" : Bool;
      "FIT-506 LOW_SET VALIDATION TIME OVER_(SYSTEM STOP)" : Bool;
      "EDI-501A PRODUCT OUT PRESSURE FIT-506 HIGH" : Bool;
      "FIT-506 HIGH_SET VALIDATION TIME OVER_(SYSTEM STOP)" : Bool;
      "EDI-501B CONCENTRATE OUT PRESSURE FIT-507 LOW" : Bool;
      "FIT-507 LOW_SET VALIDATION TIME OVER_(SYSTEM STOP)" : Bool;
      "EDI-501B CONCENTRATE OUT PRESSURE FIT-507 HIGH" : Bool;
      "FIT-507 HIGH_SET VALIDATION TIME OVER_(SYSTEM STOP)" : Bool;
      "EDI-501A PRODUCT OUT PRESSURE FIT-508 LOW" : Bool;
      "FIT-508 LOW_SET VALIDATION TIME OVER_(SYSTEM STOP)" : Bool;
      "EDI-501A PRODUCT OUT PRESSURE FIT-508 HIGH" : Bool;
      "FIT-508 HIGH_SET VALIDATION TIME OVER_(SYSTEM STOP)" : Bool;
   END_VAR
BEGIN
END_DATA_BLOCK

DATA_BLOCK "P_TRIG"   // DB98
{ S7_Optimized_Access := 'TRUE' }
// stored: MemoryReserve 100
   VAR
      ARR : Array[0..150] of Bool;
   END_VAR
BEGIN
END_DATA_BLOCK

DATA_BLOCK "INTERLOCK DB"   // DB70
{ S7_Optimized_Access := 'FALSE' }
   VAR
      "RO-1 SET PARAMETER" : Struct
         "ORP-301 HH" : Real;
         "ORP-301 H" : Real;
         "pH-301 HIGH" : Real;
         "pH-301 LOW" : Real;
         "pH-302 HIGH" : Real;
         "pH-302 LOW" : Real;
         "CT-301 H" : Real;
         "CT-301 HH" : Real;
         "CT-302 H" : Real;
         "CT-302 HH" : Real;
      END_STRUCT;
      "RO-1 PARAMETER BUFF" : Struct
         "ORP-301 BUFF" : Int;
         "pH-301 BUFF" : Int;
         "pH-302 BUFF" : Int;
         "CT-301 BUFF" : Int;
         "CT-302 BUFF" : Int;
      END_STRUCT;
      "RO-1 SET TIMER" : Struct
         "LPS-301 TIMER SET" : Int;
         "LPS-302 TIMER SET" : Int;
         "HPS-301 TIMER SET" : Int;
         "HPS-302 TIMER SET" : Int;
         "ORP-301 TIMER SET" : Int;
         "CT-301 HIGH TIMER SET" : Int;
         "CT-302 HIGH TIMER SET" : Int;
         "AGLV-301A FLUSH TIME SET" : Int;
         "AGLV-301B FLUSH  TIME SET" : Int;
      END_STRUCT;
      "RO-1 PV TIMER" : Struct
         "LPS-301 TIMER PV" : Int;
         "LPS-302 TIMER PV" : Int;
         "HPS-301 TIMER PV" : Int;
         "HPS-302 TIMER PV" : Int;
         "ORP-301 TIMER PV" : Int;
         "CT-301 HIGH TIMER PV" : Int;
         "CT-302 HIGH TIMER PV" : Int;
         "AGLV-301A FLUSH TIME PV" : Int;
         "AGLV-301B FLUSH  TIME PV" : Int;
      END_STRUCT;
      "RO-2 SET PARAMETER" : Struct
         "pH-401 HIGH" : Real;
         "pH-401 LOW" : Real;
         "pH-402 HIGH" : Real;
         "pH-402 LOW" : Real;
         "CT-401 H" : Real;
         "CT-401 HH" : Real;
         "CT-402 H" : Real;
         "CT-402 HH" : Real;
      END_STRUCT;
      "RO-2 PARAMETER BUFF" : Struct
         "pH-401 BUFF" : Int;
         "pH-402 BUFF" : Int;
         "CT-401 BUFF" : Int;
         "CT-402 BUFF" : Int;
      END_STRUCT;
      "RO-2 SET TIMER" : Struct
         "LPS-401 TIMER SET" : Int;
         "LPS-402 TIMER SET" : Int;
         "HPS-401 TIMER SET" : Int;
         "HPS-402 TIMER SET" : Int;
         "CT-401 HIGH TIMER SET" : Int;
         "CT-402 HIGH TIMER SET" : Int;
         "AGLV-401A FLUSH TIME SET" : Int;
         "AGLV-401B FLUSH  TIME SET" : Int;
      END_STRUCT;
      "RO-2 PV TIMER" : Struct
         "LPS-401 TIMER PV" : Int;
         "LPS-402 TIMER PV" : Int;
         "HPS-401 TIMER PV" : Int;
         "HPS-402 TIMER PV" : Int;
         "CT-401 HIGH TIMER PV" : Int;
         "CT-402 HIGH TIMER PV" : Int;
         "AGLV-401A FLUSH TIME PV" : Int;
         "AGLV-401B FLUSH  TIME PV" : Int;
      END_STRUCT;
      "EDI SET PARAMETER" : Struct
         "PT-501 LOW" : Real;
         "PT-501 HIGH" : Real;
         "PT-502 LOW" : Real;
         "PT-502 HIGH" : Real;
         "PT-503 HIGH" : Real;
         "PT-504 HIGH" : Real;
         "PT-505 HIGH" : Real;
         "PT-506 HIGH" : Real;
         "FIT-501 LOW" : Real;
         "FIT-502 LOW" : Real;
         "FIT-503 LOW" : Real;
         "FIT-504 LOW" : Real;
         "FIT-505 LOW" : Real;
         "FIT-505 HIGH" : Real;
         "FIT-506 LOW" : Real;
         "FIT-506 HIGH" : Real;
         "FIT-507 LOW" : Real;
         "FIT-507 HIGH" : Real;
         "FIT-508 LOW" : Real;
         "FIT-508 HIGH" : Real;
         "pHIT-501 - LOW" : Real;
         "pHIT-501 - High" : Real;
         "pHIT-502 - LOW" : Real;
         "pHIT-502 - High" : Real;
         "RIT-501 HIGH" : Real;
         "RIT-502 HIGH" : Real;
         "RIT-501 LOW" : Real;
         "RIT-502 LOW" : Real;
      END_STRUCT;
      "EDI PARAMETER BUFF" : Struct
         "PT-501 LOW/ HIGH BUFF" : Int;
         "PT-502 LOW / HIGH BUFF" : Int;
         "PT-503 HIGH" : Int;
         "PT-504 HIGH" : Int;
         "PT-505 HIGH" : Int;
         "PT-506 HIGH" : Int;
         "FIT-501 LOW BUFF" : Int;
         "FIT-502 LOW  BUFF" : Int;
         "FIT-503 LOW BUFF" : Int;
         "FIT-504 LOW BUFF" : Int;
         "FIT-505 LOW / HIGH BUFF" : Int;
         "FIT-506 LOW / HIGH BUFF" : Int;
         "FIT-507 LOW / HIGH BUFF" : Int;
         "FIT-508 LOW / HIGH BUFF" : Int;
         "pHIT-501 - LOW / High BUFF" : Int;
         "pHIT-502 - LOW / High BUFF" : Int;
         "RIT-501 HIGH/LOW BUFF" : Int;
         "RIT-502 HIGH/ LOW BUFF" : Int;
      END_STRUCT;
      "EDI SET TIMER" : Struct
         "PT-501 LOW TIMER SET" : Int;
         "PT-501 HIGH TIMER SET" : Int;
         "PT-502 LOW TIMER SET" : Int;
         "PT-502 HIGH TIMER SET" : Int;
         "PT-503 HIGH TIMER SET" : Int;
         "PT-504 HIGH TIMER SET" : Int;
         "PT-505 HIGH TIMER SET" : Int;
         "PT-506 HIGH TIMER SET" : Int;
         "FIT-501 LOW TIMER SET" : Int;
         "FIT-502 LOW TIMER SET" : Int;
         "FIT-503 LOW TIMER SET" : Int;
         "FIT-504 LOW TIMER SET" : Int;
         "FIT-505 LOW TIMER SET" : Int;
         "FIT-505 HIGH TIMER SET" : Int;
         "FIT-506 LOW TIMER SET" : Int;
         "FIT-506 HIGH TIMER SET" : Int;
         "FIT-507 LOW TIMER SET" : Int;
         "FIT-507 HIGH TIMER SET" : Int;
         "FIT-508 LOW TIMER SET" : Int;
         "FIT-508 HIGH TIMER SET" : Int;
         "pHIT-501 - LOW TIMER SET" : Int;
         "pHIT-501 - High TIMER SET" : Int;
         "pHIT-502 - LOW TIMER SET" : Int;
         "pHIT-502 - High TIMER SET" : Int;
         "RIT-501 HIGH TIMER SET" : Int;
         "RIT-502 HIGH TIMER SET" : Int;
      END_STRUCT;
      "EDI PV TIMER" : Struct
         "PT-501 LOW TIMER PV" : Int;
         "PT-501 HIGH TIMER PV" : Int;
         "PT-502 LOW TIMER PV" : Int;
         "PT-502 HIGH TIMER PV" : Int;
         "PT-503 HIGH TIMER PV" : Int;
         "PT-504 HIGH TIMER PV" : Int;
         "PT-505 HIGH TIMER PV" : Int;
         "PT-506 HIGH TIMER PV" : Int;
         "FIT-501 LOW TIMER PV" : Int;
         "FIT-502 LOW TIMER PV" : Int;
         "FIT-503 LOW TIMER PV" : Int;
         "FIT-504 LOW TIMER PV" : Int;
         "FIT-505 LOW TIMER PV" : Int;
         "FIT-505 HIGH TIMER PV" : Int;
         "FIT-506 LOW TIMER PV" : Int;
         "FIT-506 HIGH TIMER PV" : Int;
         "FIT-507 LOW TIMER PV" : Int;
         "FIT-507 HIGH TIMER PV" : Int;
         "FIT-508 LOW TIMER PV" : Int;
         "FIT-508 HIGH TIMER PV" : Int;
         "pHIT-501 - LOW TIMER PV" : Int;
         "pHIT-501 - High TIMER PV" : Int;
         "pHIT-502 - LOW TIMER PV" : Int;
         "pHIT-502 - High TIMER PV" : Int;
         "RIT-501 HIGH TIMER PV" : Int;
         "RIT-502 HIGH TIMER PV" : Int;
      END_STRUCT;
   END_VAR
BEGIN
END_DATA_BLOCK

DATA_BLOCK "EDI DB"   // DB111
{ S7_Optimized_Access := 'FALSE' }
   VAR
      "EDI FEED PUMP 401ABC" : Bool;
      "EDI 501A" : Bool;
      "EDI 501B" : Bool;
      "AGLV-501 BUFF" : Int;
      "LEVEL HI RECIRC BUFF" : Int;
      "AGLV-501" : Bool;
      "AGLV-502" : Bool;
      "FLUSHING TIMER SET" : Int;
      "FLUSHING TIMER PV" : Int;
      "RECIRCULATION ON TIMER SET" : Int;
      "RECIRCULATION ON TIMER PV" : Int;
      "RECIRCULATION OFF TIMER SET" : Int;
      "RECIRCULATION OFF TIMER PV" : Int;
      "AGLV 501 FOR FLUSHING" : Bool;
      "AGLV 501 FOR RECIRCULATION" : Bool;
   END_VAR
BEGIN
END_DATA_BLOCK

DATA_BLOCK "RO 1 LEVEL DB"   // DB199
{ S7_Optimized_Access := 'FALSE' }
   VAR
      "AGLV 301 BUFF" : Int;
      "RECIRCULATION TIME SV" : Int;
      "RECIRCULATION TIME PV" : Int;
      "AGLV 302 BUFF" : Int;
      "RECIRCULATION TIME 302 SV" : Int;
      "RECIRCULATION TIME 302 PV" : Int;
      "LEVEL HI RECIRC BUFF" : Int;
      "LEVEL HI RECIRC RO ON TIME SV" : Int;
      "LEVEL HI RECIRC RO ON TIME PV" : Int;
      "LEVEL HI RECIRC RO OFF TIME SV" : Int;
      "LEVEL HI RECIRC RO OFF TIME PV" : Int;
   END_VAR
BEGIN
END_DATA_BLOCK

DATA_BLOCK "RO_1 DB"   // DB72
{ S7_Optimized_Access := 'FALSE' }
   VAR RETAIN
      OUTPUT : Struct
         "ABV-301" : Bool;
         "ABV-302" : Bool;
         "AGLV-301" : Bool;
         "AGLV-302" : Bool;
         "DP-703" : Bool;
         "DP-704" : Bool;
         "DP-705" : Bool;
         "RO-1 FEED PUMP" : Bool;
         "RO-1 HPP-301A" : Bool;
         "RO-1 HPP-301B" : Bool;
         "AGLV-301 RECIRC" : Bool;
         "AGLV-302 RECIRC" : Bool;
      END_STRUCT;
   END_VAR
BEGIN
END_DATA_BLOCK

DATA_BLOCK "RO_2 DB"   // DB102
{ S7_Optimized_Access := 'FALSE' }
   VAR
      "RO-2 P-401A/B/C FEED PUMP" : Bool;
      "HPP-402 A" : Bool;
      "HPP-402 B" : Bool;
      "AGLV-401 RECIRC" : Bool;
      "AGLV-402 RECIRC" : Bool;
      "AGLV-401" : Bool;
      "AGLV-402" : Bool;
   END_VAR
BEGIN
END_DATA_BLOCK

DATA_BLOCK "RO_2_LEVEL DB"   // DB210
{ S7_Optimized_Access := 'FALSE' }
   VAR
      "AGLV 401 BUFF" : Int;
      "RECIRCULATION TIME SV" : Int;
      "RECIRCULATION TIME PV" : Int;
      "AGLV 402 BUFF" : Int;
      "RECIRCULATION TIME 402 SV" : Int;
      "RECIRCULATION TIME 402 PV" : Int;
      "LEVEL HI RECIRC BUFF" : Int;
      "LEVEL HI RECIRC RO ON TIME SV" : Int;
      "LEVEL HI RECIRC RO ON TIME PV" : Int;
      "LEVEL HI RECIRC RO OFF TIME SV" : Int;
      "LEVEL HI RECIRC RO OFF TIME PV" : Int;
   END_VAR
BEGIN
END_DATA_BLOCK

ORGANIZATION_BLOCK "Main"   // OB1, LAD, ProgramCycle
TITLE = "Main Program Sweep (Cycle)"
{ S7_Optimized_Access := 'TRUE' }
// stored: SetENOAutomatically false
   VAR_INPUT
      Initial_Call : Bool;   // Initial call of this OB
      Remanence : Bool;   // =True, if remanent data are available
   END_VAR
   VAR_TEMP   // added for the SCL form of the ladder/FBD networks
      _w1 : Bool;
      _w2 : Bool;
      _w3 : Bool;
      _w4 : Bool;
      _w5 : Bool;
      _w6 : Bool;
      _w7 : Bool;
      _w8 : Bool;
      _w9 : Bool;
      _w10 : Bool;
      _w11 : Bool;
      _w12 : Bool;
      _w13 : Bool;
      _w14 : Bool;
      _w15 : Bool;
      _w16 : Bool;
      _w17 : Bool;
      _w18 : Bool;
      _w19 : Bool;
      _w20 : Bool;
   END_VAR
BEGIN

REGION Network 1
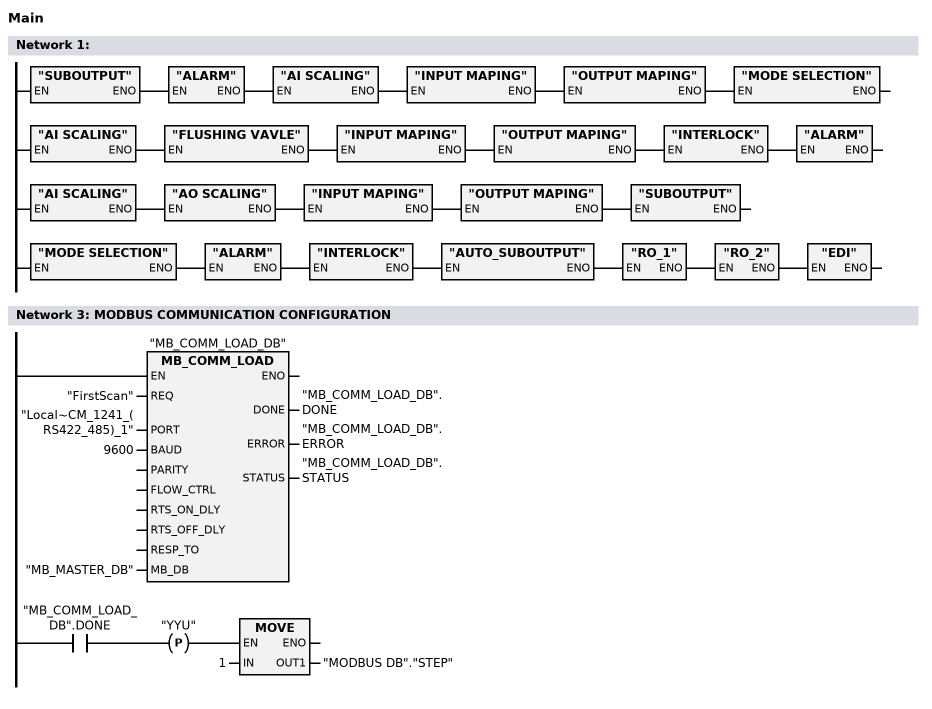
   RUNG wire#powerrail
      "SUBOUTPUT"()
      "ALARM"()
      "AI SCALING"()
      "INPUT MAPING"()
      "OUTPUT MAPING"()
      "MODE SELECTION"()
   END_RUNG
   RUNG wire#powerrail
      "AI SCALING"()
      "FLUSHING VAVLE"()
      "INPUT MAPING"()
      "OUTPUT MAPING"()
      "INTERLOCK"()
      "ALARM"()
   END_RUNG
   RUNG wire#powerrail
      "AI SCALING"()
      "AO SCALING"()
      "INPUT MAPING"()
      "OUTPUT MAPING"()
      "SUBOUTPUT"()
   END_RUNG
   RUNG wire#powerrail
      "MODE SELECTION"()
      "ALARM"()
      "INTERLOCK"()
      "AUTO_SUBOUTPUT"()
      "RO_1"()
      "RO_2"()
      "EDI"()
   END_RUNG
   // the same network as SCL:
   "SUBOUTPUT"(ENO => #_w1);
   "ALARM"(EN := #_w1, ENO => #_w2);
   "AI SCALING"(EN := #_w2, ENO => #_w3);
   "INPUT MAPING"(EN := #_w3, ENO => #_w4);
   "OUTPUT MAPING"(EN := #_w4, ENO => #_w5);
   IF #_w5 THEN "MODE SELECTION"(); END_IF;
   "AI SCALING"(ENO => #_w6);
   "FLUSHING VAVLE"(EN := #_w6, ENO => #_w7);
   "INPUT MAPING"(EN := #_w7, ENO => #_w8);
   "OUTPUT MAPING"(EN := #_w8, ENO => #_w9);
   "INTERLOCK"(EN := #_w9, ENO => #_w10);
   IF #_w10 THEN "ALARM"(); END_IF;
   "AI SCALING"(ENO => #_w11);
   "AO SCALING"(EN := #_w11, ENO => #_w12);
   "INPUT MAPING"(EN := #_w12, ENO => #_w13);
   "OUTPUT MAPING"(EN := #_w13, ENO => #_w14);
   IF #_w14 THEN "SUBOUTPUT"(); END_IF;
   "MODE SELECTION"(ENO => #_w15);
   "ALARM"(EN := #_w15, ENO => #_w16);
   "INTERLOCK"(EN := #_w16, ENO => #_w17);
   "AUTO_SUBOUTPUT"(EN := #_w17, ENO => #_w18);
   "RO_1"(EN := #_w18, ENO => #_w19);
   "RO_2"(EN := #_w19, ENO => #_w20);
   IF #_w20 THEN "EDI"(); END_IF;
END_REGION

REGION Network 3: MODBUS COMMUNICATION CONFIGURATION
   RUNG wire#powerrail
      "MB_COMM_LOAD_DB".MB_COMM_LOAD(REQ := "FirstScan", PORT := "Local~CM_1241_(RS422_485)_1", BAUD := 9600, PARITY :=, FLOW_CTRL :=, RTS_ON_DLY :=, RTS_OFF_DLY :=, RESP_TO :=, MB_DB := "MB_MASTER_DB", DONE => "MB_COMM_LOAD_DB".DONE, ERROR => "MB_COMM_LOAD_DB".ERROR, STATUS => "MB_COMM_LOAD_DB".STATUS)
   END_RUNG
   RUNG wire#powerrail
      Contact( "MB_COMM_LOAD_DB".DONE )
      P_Trig( "YYU" )
      Move(in := 1, out1 => "MODBUS DB"."STEP")
   END_RUNG
   // the same network as SCL:
   "MB_COMM_LOAD_DB"(REQ := "FirstScan",   // MB_COMM_LOAD
                     PORT := "Local~CM_1241_(RS422_485)_1",
                     BAUD := 9600,
                     MB_DB := "MB_MASTER_DB",
                     DONE => "MB_COMM_LOAD_DB".DONE,
                     ERROR => "MB_COMM_LOAD_DB".ERROR,
                     STATUS => "MB_COMM_LOAD_DB".STATUS);
   #_w1 := "MB_COMM_LOAD_DB".DONE AND NOT "YYU";   // rising edge
   "YYU" := "MB_COMM_LOAD_DB".DONE;
   IF #_w1 THEN "MODBUS DB"."STEP" := 1; END_IF;
END_REGION

REGION Network 4: slave plc
END_REGION
END_ORGANIZATION_BLOCK

FUNCTION "SUBOUTPUT" : Void   // FC4, LAD
{ S7_Optimized_Access := 'TRUE' }
// stored: SetENOAutomatically false
BEGIN

REGION Network 1: P-202 A RO 1 FEED PUMP
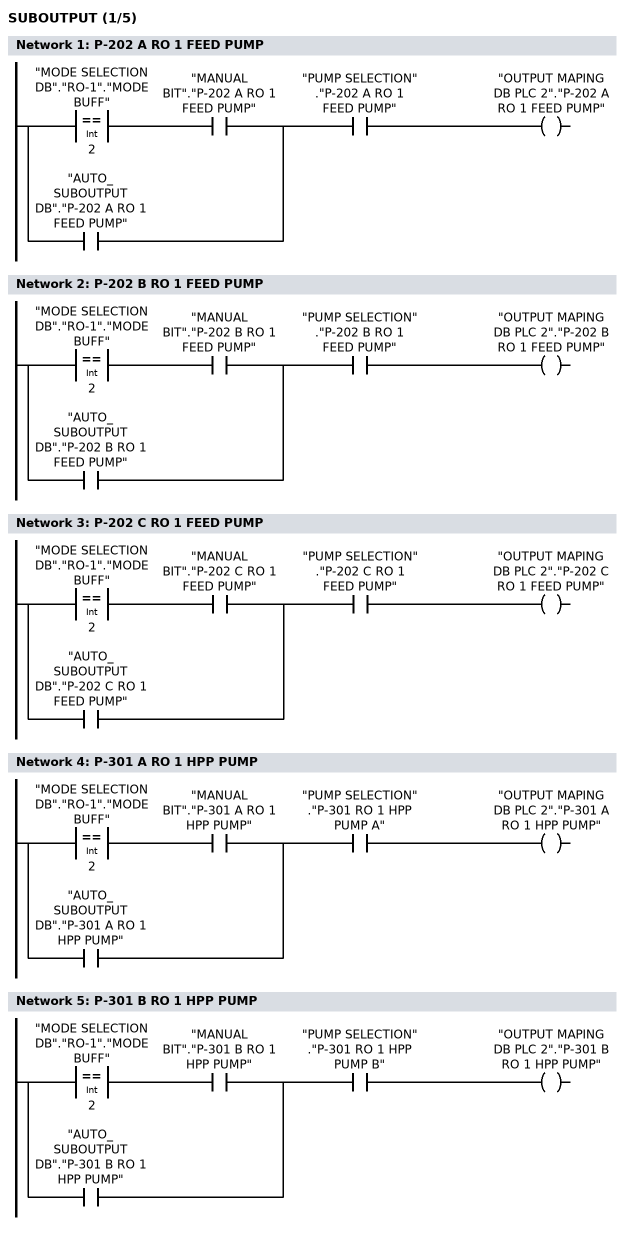
   RUNG wire#powerrail
      { S7_Templates := "SrcType := Int" } EQ_Contact(in1 := "MODE SELECTION DB"."RO-1"."MODE BUFF", in2 := 2)
      Contact( "MANUAL BIT"."P-202 A RO 1 FEED PUMP" )
      wire#w1
      Contact( "PUMP SELECTION"."P-202 A RO 1 FEED PUMP" )
      Coil( "OUTPUT MAPING DB PLC 2"."P-202 A RO 1 FEED PUMP" )
   END_RUNG
   RUNG wire#powerrail
      Contact( "AUTO_SUBOUTPUT DB"."P-202 A RO 1 FEED PUMP" )
   END_RUNG wire#w1
   // the same network as SCL:
   "OUTPUT MAPING DB PLC 2"."P-202 A RO 1 FEED PUMP" := ((("MODE SELECTION DB"."RO-1"."MODE BUFF" = 2) AND "MANUAL BIT"."P-202 A RO 1 FEED PUMP") OR "AUTO_SUBOUTPUT DB"."P-202 A RO 1 FEED PUMP") AND "PUMP SELECTION"."P-202 A RO 1 FEED PUMP";
END_REGION

REGION Network 2: P-202 B RO 1 FEED PUMP
   RUNG wire#powerrail
      { S7_Templates := "SrcType := Int" } EQ_Contact(in1 := "MODE SELECTION DB"."RO-1"."MODE BUFF", in2 := 2)
      Contact( "MANUAL BIT"."P-202 B RO 1 FEED PUMP" )
      wire#w1
      Contact( "PUMP SELECTION"."P-202 B RO 1 FEED PUMP" )
      Coil( "OUTPUT MAPING DB PLC 2"."P-202 B RO 1 FEED PUMP" )
   END_RUNG
   RUNG wire#powerrail
      Contact( "AUTO_SUBOUTPUT DB"."P-202 B RO 1 FEED PUMP" )
   END_RUNG wire#w1
   // the same network as SCL:
   "OUTPUT MAPING DB PLC 2"."P-202 B RO 1 FEED PUMP" := ((("MODE SELECTION DB"."RO-1"."MODE BUFF" = 2) AND "MANUAL BIT"."P-202 B RO 1 FEED PUMP") OR "AUTO_SUBOUTPUT DB"."P-202 B RO 1 FEED PUMP") AND "PUMP SELECTION"."P-202 B RO 1 FEED PUMP";
END_REGION

REGION Network 3: P-202 C RO 1 FEED PUMP
   RUNG wire#powerrail
      { S7_Templates := "SrcType := Int" } EQ_Contact(in1 := "MODE SELECTION DB"."RO-1"."MODE BUFF", in2 := 2)
      Contact( "MANUAL BIT"."P-202 C RO 1 FEED PUMP" )
      wire#w1
      Contact( "PUMP SELECTION"."P-202 C RO 1 FEED PUMP" )
      Coil( "OUTPUT MAPING DB PLC 2"."P-202 C RO 1 FEED PUMP" )
   END_RUNG
   RUNG wire#powerrail
      Contact( "AUTO_SUBOUTPUT DB"."P-202 C RO 1 FEED PUMP" )
   END_RUNG wire#w1
   // the same network as SCL:
   "OUTPUT MAPING DB PLC 2"."P-202 C RO 1 FEED PUMP" := ((("MODE SELECTION DB"."RO-1"."MODE BUFF" = 2) AND "MANUAL BIT"."P-202 C RO 1 FEED PUMP") OR "AUTO_SUBOUTPUT DB"."P-202 C RO 1 FEED PUMP") AND "PUMP SELECTION"."P-202 C RO 1 FEED PUMP";
END_REGION

REGION Network 4: P-301 A RO 1 HPP PUMP
   RUNG wire#powerrail
      { S7_Templates := "SrcType := Int" } EQ_Contact(in1 := "MODE SELECTION DB"."RO-1"."MODE BUFF", in2 := 2)
      Contact( "MANUAL BIT"."P-301 A RO 1 HPP PUMP" )
      wire#w1
      Contact( "PUMP SELECTION"."P-301 RO 1 HPP PUMP A" )
      Coil( "OUTPUT MAPING DB PLC 2"."P-301 A RO 1 HPP PUMP" )
   END_RUNG
   RUNG wire#powerrail
      Contact( "AUTO_SUBOUTPUT DB"."P-301 A RO 1 HPP PUMP" )
   END_RUNG wire#w1
   // the same network as SCL:
   "OUTPUT MAPING DB PLC 2"."P-301 A RO 1 HPP PUMP" := ((("MODE SELECTION DB"."RO-1"."MODE BUFF" = 2) AND "MANUAL BIT"."P-301 A RO 1 HPP PUMP") OR "AUTO_SUBOUTPUT DB"."P-301 A RO 1 HPP PUMP") AND "PUMP SELECTION"."P-301 RO 1 HPP PUMP A";
END_REGION

REGION Network 5: P-301 B RO 1 HPP PUMP
   RUNG wire#powerrail
      { S7_Templates := "SrcType := Int" } EQ_Contact(in1 := "MODE SELECTION DB"."RO-1"."MODE BUFF", in2 := 2)
      Contact( "MANUAL BIT"."P-301 B RO 1 HPP PUMP" )
      wire#w1
      Contact( "PUMP SELECTION"."P-301 RO 1 HPP PUMP B" )
      Coil( "OUTPUT MAPING DB PLC 2"."P-301 B RO 1 HPP PUMP" )
   END_RUNG
   RUNG wire#powerrail
      Contact( "AUTO_SUBOUTPUT DB"."P-301 B RO 1 HPP PUMP" )
   END_RUNG wire#w1
   // the same network as SCL:
   "OUTPUT MAPING DB PLC 2"."P-301 B RO 1 HPP PUMP" := ((("MODE SELECTION DB"."RO-1"."MODE BUFF" = 2) AND "MANUAL BIT"."P-301 B RO 1 HPP PUMP") OR "AUTO_SUBOUTPUT DB"."P-301 B RO 1 HPP PUMP") AND "PUMP SELECTION"."P-301 RO 1 HPP PUMP B";
END_REGION

REGION Network 6: P-401 A RO 2 FEED PUMP
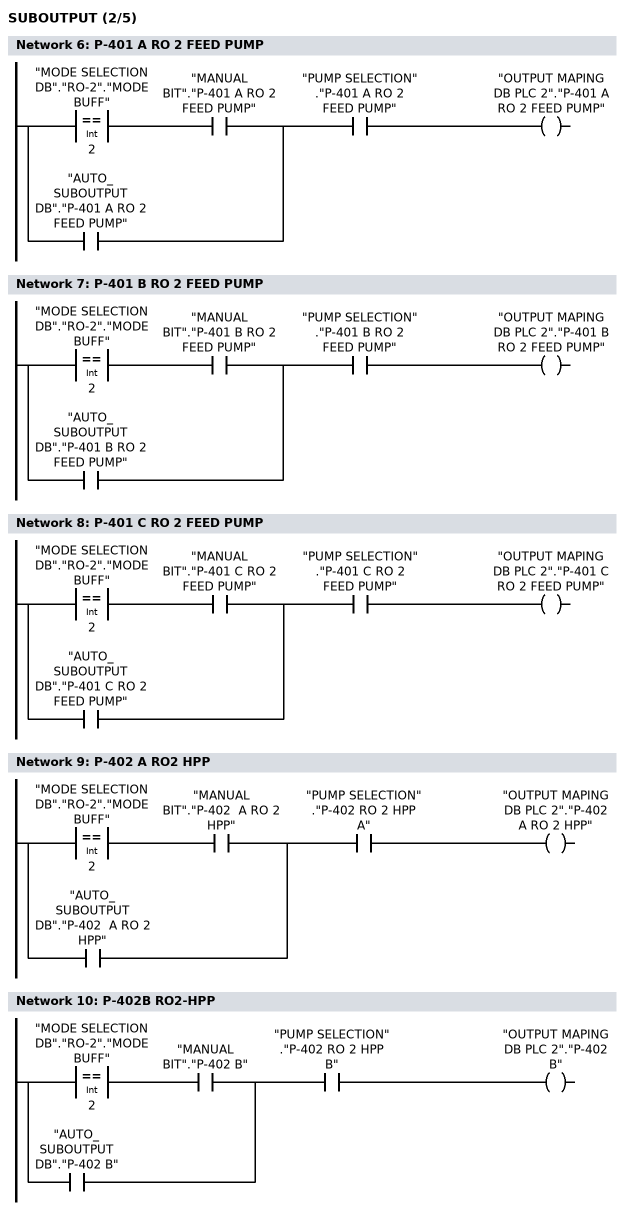
   RUNG wire#powerrail
      { S7_Templates := "SrcType := Int" } EQ_Contact(in1 := "MODE SELECTION DB"."RO-2"."MODE BUFF", in2 := 2)
      Contact( "MANUAL BIT"."P-401 A RO 2 FEED PUMP" )
      wire#w1
      Contact( "PUMP SELECTION"."P-401 A RO 2 FEED PUMP" )
      Coil( "OUTPUT MAPING DB PLC 2"."P-401 A RO 2 FEED PUMP" )
   END_RUNG
   RUNG wire#powerrail
      Contact( "AUTO_SUBOUTPUT DB"."P-401 A RO 2 FEED PUMP" )
   END_RUNG wire#w1
   // the same network as SCL:
   "OUTPUT MAPING DB PLC 2"."P-401 A RO 2 FEED PUMP" := ((("MODE SELECTION DB"."RO-2"."MODE BUFF" = 2) AND "MANUAL BIT"."P-401 A RO 2 FEED PUMP") OR "AUTO_SUBOUTPUT DB"."P-401 A RO 2 FEED PUMP") AND "PUMP SELECTION"."P-401 A RO 2 FEED PUMP";
END_REGION

REGION Network 7: P-401 B RO 2 FEED PUMP
   RUNG wire#powerrail
      { S7_Templates := "SrcType := Int" } EQ_Contact(in1 := "MODE SELECTION DB"."RO-2"."MODE BUFF", in2 := 2)
      Contact( "MANUAL BIT"."P-401 B RO 2 FEED PUMP" )
      wire#w1
      Contact( "PUMP SELECTION"."P-401 B RO 2 FEED PUMP" )
      Coil( "OUTPUT MAPING DB PLC 2"."P-401 B RO 2 FEED PUMP" )
   END_RUNG
   RUNG wire#powerrail
      Contact( "AUTO_SUBOUTPUT DB"."P-401 B RO 2 FEED PUMP" )
   END_RUNG wire#w1
   // the same network as SCL:
   "OUTPUT MAPING DB PLC 2"."P-401 B RO 2 FEED PUMP" := ((("MODE SELECTION DB"."RO-2"."MODE BUFF" = 2) AND "MANUAL BIT"."P-401 B RO 2 FEED PUMP") OR "AUTO_SUBOUTPUT DB"."P-401 B RO 2 FEED PUMP") AND "PUMP SELECTION"."P-401 B RO 2 FEED PUMP";
END_REGION

REGION Network 8: P-401 C RO 2 FEED PUMP
   RUNG wire#powerrail
      { S7_Templates := "SrcType := Int" } EQ_Contact(in1 := "MODE SELECTION DB"."RO-2"."MODE BUFF", in2 := 2)
      Contact( "MANUAL BIT"."P-401 C RO 2 FEED PUMP" )
      wire#w1
      Contact( "PUMP SELECTION"."P-401 C RO 2 FEED PUMP" )
      Coil( "OUTPUT MAPING DB PLC 2"."P-401 C RO 2 FEED PUMP" )
   END_RUNG
   RUNG wire#powerrail
      Contact( "AUTO_SUBOUTPUT DB"."P-401 C RO 2 FEED PUMP" )
   END_RUNG wire#w1
   // the same network as SCL:
   "OUTPUT MAPING DB PLC 2"."P-401 C RO 2 FEED PUMP" := ((("MODE SELECTION DB"."RO-2"."MODE BUFF" = 2) AND "MANUAL BIT"."P-401 C RO 2 FEED PUMP") OR "AUTO_SUBOUTPUT DB"."P-401 C RO 2 FEED PUMP") AND "PUMP SELECTION"."P-401 C RO 2 FEED PUMP";
END_REGION

REGION Network 9: P-402 A RO2 HPP
   RUNG wire#powerrail
      { S7_Templates := "SrcType := Int" } EQ_Contact(in1 := "MODE SELECTION DB"."RO-2"."MODE BUFF", in2 := 2)
      Contact( "MANUAL BIT"."P-402  A RO 2 HPP" )
      wire#w1
      Contact( "PUMP SELECTION"."P-402 RO 2 HPP A" )
      Coil( "OUTPUT MAPING DB PLC 2"."P-402  A RO 2 HPP" )
   END_RUNG
   RUNG wire#powerrail
      Contact( "AUTO_SUBOUTPUT DB"."P-402  A RO 2 HPP" )
   END_RUNG wire#w1
   // the same network as SCL:
   "OUTPUT MAPING DB PLC 2"."P-402  A RO 2 HPP" := ((("MODE SELECTION DB"."RO-2"."MODE BUFF" = 2) AND "MANUAL BIT"."P-402  A RO 2 HPP") OR "AUTO_SUBOUTPUT DB"."P-402  A RO 2 HPP") AND "PUMP SELECTION"."P-402 RO 2 HPP A";
END_REGION

REGION Network 10: P-402B RO2-HPP
   RUNG wire#powerrail
      { S7_Templates := "SrcType := Int" } EQ_Contact(in1 := "MODE SELECTION DB"."RO-2"."MODE BUFF", in2 := 2)
      Contact( "MANUAL BIT"."P-402 B" )
      wire#w1
      Contact( "PUMP SELECTION"."P-402 RO 2 HPP B" )
      Coil( "OUTPUT MAPING DB PLC 2"."P-402 B" )
   END_RUNG
   RUNG wire#powerrail
      Contact( "AUTO_SUBOUTPUT DB"."P-402 B" )
   END_RUNG wire#w1
   // the same network as SCL:
   "OUTPUT MAPING DB PLC 2"."P-402 B" := ((("MODE SELECTION DB"."RO-2"."MODE BUFF" = 2) AND "MANUAL BIT"."P-402 B") OR "AUTO_SUBOUTPUT DB"."P-402 B") AND "PUMP SELECTION"."P-402 RO 2 HPP B";
END_REGION

REGION Network 11: P-501 A EDI FEED PUMP
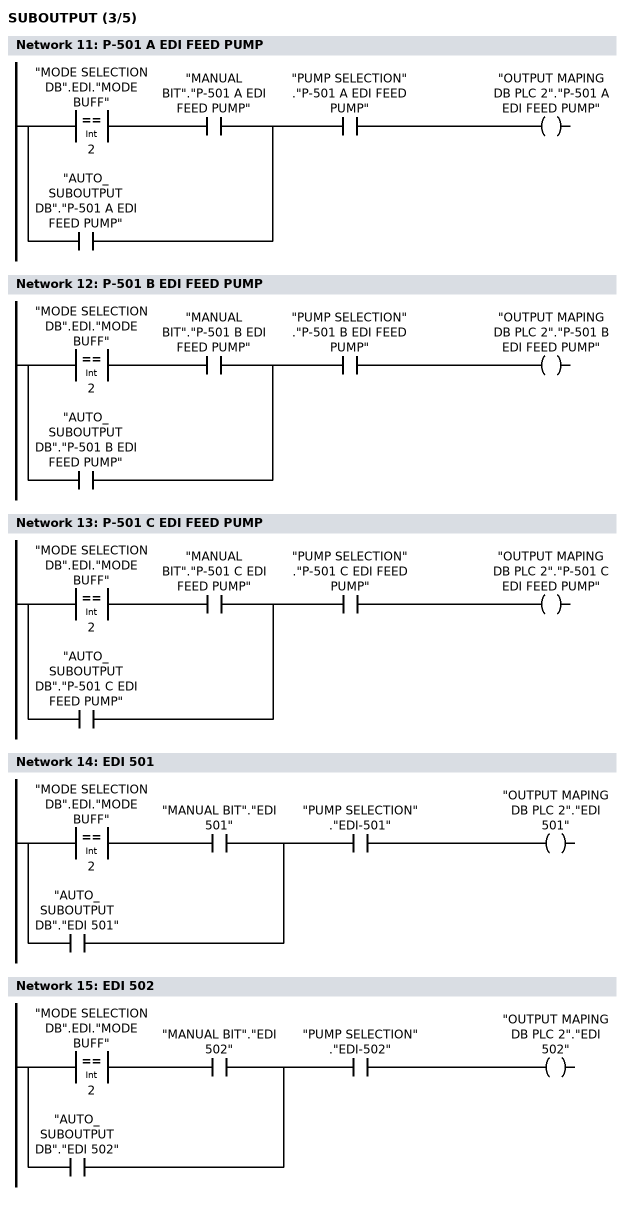
   RUNG wire#powerrail
      { S7_Templates := "SrcType := Int" } EQ_Contact(in1 := "MODE SELECTION DB".EDI."MODE BUFF", in2 := 2)
      Contact( "MANUAL BIT"."P-501 A EDI FEED PUMP" )
      wire#w1
      Contact( "PUMP SELECTION"."P-501 A EDI FEED PUMP" )
      Coil( "OUTPUT MAPING DB PLC 2"."P-501 A EDI FEED PUMP" )
   END_RUNG
   RUNG wire#powerrail
      Contact( "AUTO_SUBOUTPUT DB"."P-501 A EDI FEED PUMP" )
   END_RUNG wire#w1
   // the same network as SCL:
   "OUTPUT MAPING DB PLC 2"."P-501 A EDI FEED PUMP" := ((("MODE SELECTION DB".EDI."MODE BUFF" = 2) AND "MANUAL BIT"."P-501 A EDI FEED PUMP") OR "AUTO_SUBOUTPUT DB"."P-501 A EDI FEED PUMP") AND "PUMP SELECTION"."P-501 A EDI FEED PUMP";
END_REGION

REGION Network 12: P-501 B EDI FEED PUMP
   RUNG wire#powerrail
      { S7_Templates := "SrcType := Int" } EQ_Contact(in1 := "MODE SELECTION DB".EDI."MODE BUFF", in2 := 2)
      Contact( "MANUAL BIT"."P-501 B EDI FEED PUMP" )
      wire#w1
      Contact( "PUMP SELECTION"."P-501 B EDI FEED PUMP" )
      Coil( "OUTPUT MAPING DB PLC 2"."P-501 B EDI FEED PUMP" )
   END_RUNG
   RUNG wire#powerrail
      Contact( "AUTO_SUBOUTPUT DB"."P-501 B EDI FEED PUMP" )
   END_RUNG wire#w1
   // the same network as SCL:
   "OUTPUT MAPING DB PLC 2"."P-501 B EDI FEED PUMP" := ((("MODE SELECTION DB".EDI."MODE BUFF" = 2) AND "MANUAL BIT"."P-501 B EDI FEED PUMP") OR "AUTO_SUBOUTPUT DB"."P-501 B EDI FEED PUMP") AND "PUMP SELECTION"."P-501 B EDI FEED PUMP";
END_REGION

REGION Network 13: P-501 C EDI FEED PUMP
   RUNG wire#powerrail
      { S7_Templates := "SrcType := Int" } EQ_Contact(in1 := "MODE SELECTION DB".EDI."MODE BUFF", in2 := 2)
      Contact( "MANUAL BIT"."P-501 C EDI FEED PUMP" )
      wire#w1
      Contact( "PUMP SELECTION"."P-501 C EDI FEED PUMP" )
      Coil( "OUTPUT MAPING DB PLC 2"."P-501 C EDI FEED PUMP" )
   END_RUNG
   RUNG wire#powerrail
      Contact( "AUTO_SUBOUTPUT DB"."P-501 C EDI FEED PUMP" )
   END_RUNG wire#w1
   // the same network as SCL:
   "OUTPUT MAPING DB PLC 2"."P-501 C EDI FEED PUMP" := ((("MODE SELECTION DB".EDI."MODE BUFF" = 2) AND "MANUAL BIT"."P-501 C EDI FEED PUMP") OR "AUTO_SUBOUTPUT DB"."P-501 C EDI FEED PUMP") AND "PUMP SELECTION"."P-501 C EDI FEED PUMP";
END_REGION

REGION Network 14: EDI 501
   RUNG wire#powerrail
      { S7_Templates := "SrcType := Int" } EQ_Contact(in1 := "MODE SELECTION DB".EDI."MODE BUFF", in2 := 2)
      Contact( "MANUAL BIT"."EDI 501" )
      wire#w1
      Contact( "PUMP SELECTION"."EDI-501" )
      Coil( "OUTPUT MAPING DB PLC 2"."EDI 501" )
   END_RUNG
   RUNG wire#powerrail
      Contact( "AUTO_SUBOUTPUT DB"."EDI 501" )
   END_RUNG wire#w1
   // the same network as SCL:
   "OUTPUT MAPING DB PLC 2"."EDI 501" := ((("MODE SELECTION DB".EDI."MODE BUFF" = 2) AND "MANUAL BIT"."EDI 501") OR "AUTO_SUBOUTPUT DB"."EDI 501") AND "PUMP SELECTION"."EDI-501";
END_REGION

REGION Network 15: EDI 502
   RUNG wire#powerrail
      { S7_Templates := "SrcType := Int" } EQ_Contact(in1 := "MODE SELECTION DB".EDI."MODE BUFF", in2 := 2)
      Contact( "MANUAL BIT"."EDI 502" )
      wire#w1
      Contact( "PUMP SELECTION"."EDI-502" )
      Coil( "OUTPUT MAPING DB PLC 2"."EDI 502" )
   END_RUNG
   RUNG wire#powerrail
      Contact( "AUTO_SUBOUTPUT DB"."EDI 502" )
   END_RUNG wire#w1
   // the same network as SCL:
   "OUTPUT MAPING DB PLC 2"."EDI 502" := ((("MODE SELECTION DB".EDI."MODE BUFF" = 2) AND "MANUAL BIT"."EDI 502") OR "AUTO_SUBOUTPUT DB"."EDI 502") AND "PUMP SELECTION"."EDI-502";
END_REGION

REGION Network 16: DP 703
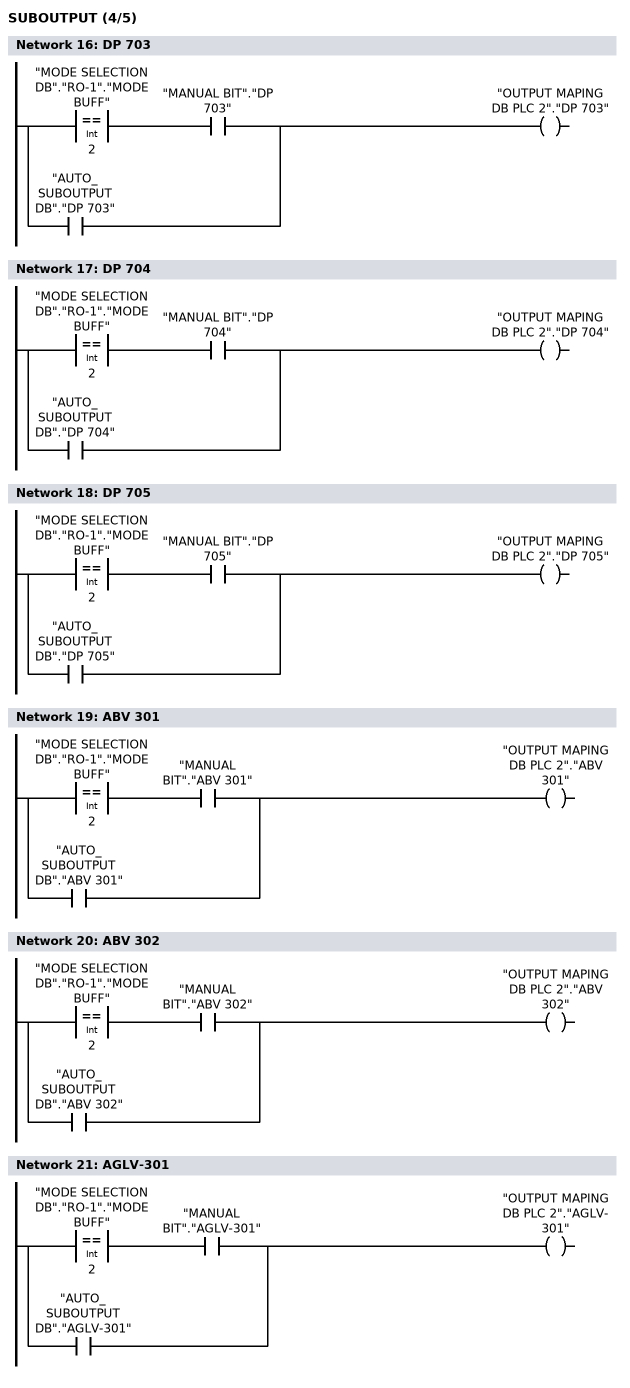
   RUNG wire#powerrail
      { S7_Templates := "SrcType := Int" } EQ_Contact(in1 := "MODE SELECTION DB"."RO-1"."MODE BUFF", in2 := 2)
      Contact( "MANUAL BIT"."DP 703" )
      wire#w1
      Coil( "OUTPUT MAPING DB PLC 2"."DP 703" )
   END_RUNG
   RUNG wire#powerrail
      Contact( "AUTO_SUBOUTPUT DB"."DP 703" )
   END_RUNG wire#w1
   // the same network as SCL:
   "OUTPUT MAPING DB PLC 2"."DP 703" := (("MODE SELECTION DB"."RO-1"."MODE BUFF" = 2) AND "MANUAL BIT"."DP 703") OR "AUTO_SUBOUTPUT DB"."DP 703";
END_REGION

REGION Network 17: DP 704
   RUNG wire#powerrail
      { S7_Templates := "SrcType := Int" } EQ_Contact(in1 := "MODE SELECTION DB"."RO-1"."MODE BUFF", in2 := 2)
      Contact( "MANUAL BIT"."DP 704" )
      wire#w1
      Coil( "OUTPUT MAPING DB PLC 2"."DP 704" )
   END_RUNG
   RUNG wire#powerrail
      Contact( "AUTO_SUBOUTPUT DB"."DP 704" )
   END_RUNG wire#w1
   // the same network as SCL:
   "OUTPUT MAPING DB PLC 2"."DP 704" := (("MODE SELECTION DB"."RO-1"."MODE BUFF" = 2) AND "MANUAL BIT"."DP 704") OR "AUTO_SUBOUTPUT DB"."DP 704";
END_REGION

REGION Network 18: DP 705
   RUNG wire#powerrail
      { S7_Templates := "SrcType := Int" } EQ_Contact(in1 := "MODE SELECTION DB"."RO-1"."MODE BUFF", in2 := 2)
      Contact( "MANUAL BIT"."DP 705" )
      wire#w1
      Coil( "OUTPUT MAPING DB PLC 2"."DP 705" )
   END_RUNG
   RUNG wire#powerrail
      Contact( "AUTO_SUBOUTPUT DB"."DP 705" )
   END_RUNG wire#w1
   // the same network as SCL:
   "OUTPUT MAPING DB PLC 2"."DP 705" := (("MODE SELECTION DB"."RO-1"."MODE BUFF" = 2) AND "MANUAL BIT"."DP 705") OR "AUTO_SUBOUTPUT DB"."DP 705";
END_REGION

REGION Network 19: ABV 301
   RUNG wire#powerrail
      { S7_Templates := "SrcType := Int" } EQ_Contact(in1 := "MODE SELECTION DB"."RO-1"."MODE BUFF", in2 := 2)
      Contact( "MANUAL BIT"."ABV 301" )
      wire#w1
      Coil( "OUTPUT MAPING DB PLC 2"."ABV 301" )
   END_RUNG
   RUNG wire#powerrail
      Contact( "AUTO_SUBOUTPUT DB"."ABV 301" )
   END_RUNG wire#w1
   // the same network as SCL:
   "OUTPUT MAPING DB PLC 2"."ABV 301" := (("MODE SELECTION DB"."RO-1"."MODE BUFF" = 2) AND "MANUAL BIT"."ABV 301") OR "AUTO_SUBOUTPUT DB"."ABV 301";
END_REGION

REGION Network 20: ABV 302
   RUNG wire#powerrail
      { S7_Templates := "SrcType := Int" } EQ_Contact(in1 := "MODE SELECTION DB"."RO-1"."MODE BUFF", in2 := 2)
      Contact( "MANUAL BIT"."ABV 302" )
      wire#w1
      Coil( "OUTPUT MAPING DB PLC 2"."ABV 302" )
   END_RUNG
   RUNG wire#powerrail
      Contact( "AUTO_SUBOUTPUT DB"."ABV 302" )
   END_RUNG wire#w1
   // the same network as SCL:
   "OUTPUT MAPING DB PLC 2"."ABV 302" := (("MODE SELECTION DB"."RO-1"."MODE BUFF" = 2) AND "MANUAL BIT"."ABV 302") OR "AUTO_SUBOUTPUT DB"."ABV 302";
END_REGION

REGION Network 21: AGLV-301
   RUNG wire#powerrail
      { S7_Templates := "SrcType := Int" } EQ_Contact(in1 := "MODE SELECTION DB"."RO-1"."MODE BUFF", in2 := 2)
      Contact( "MANUAL BIT"."AGLV-301" )
      wire#w1
      Coil( "OUTPUT MAPING DB PLC 2"."AGLV-301" )
   END_RUNG
   RUNG wire#powerrail
      Contact( "AUTO_SUBOUTPUT DB"."AGLV-301" )
   END_RUNG wire#w1
   // the same network as SCL:
   "OUTPUT MAPING DB PLC 2"."AGLV-301" := (("MODE SELECTION DB"."RO-1"."MODE BUFF" = 2) AND "MANUAL BIT"."AGLV-301") OR "AUTO_SUBOUTPUT DB"."AGLV-301";
END_REGION

REGION Network 22: AGLV-302
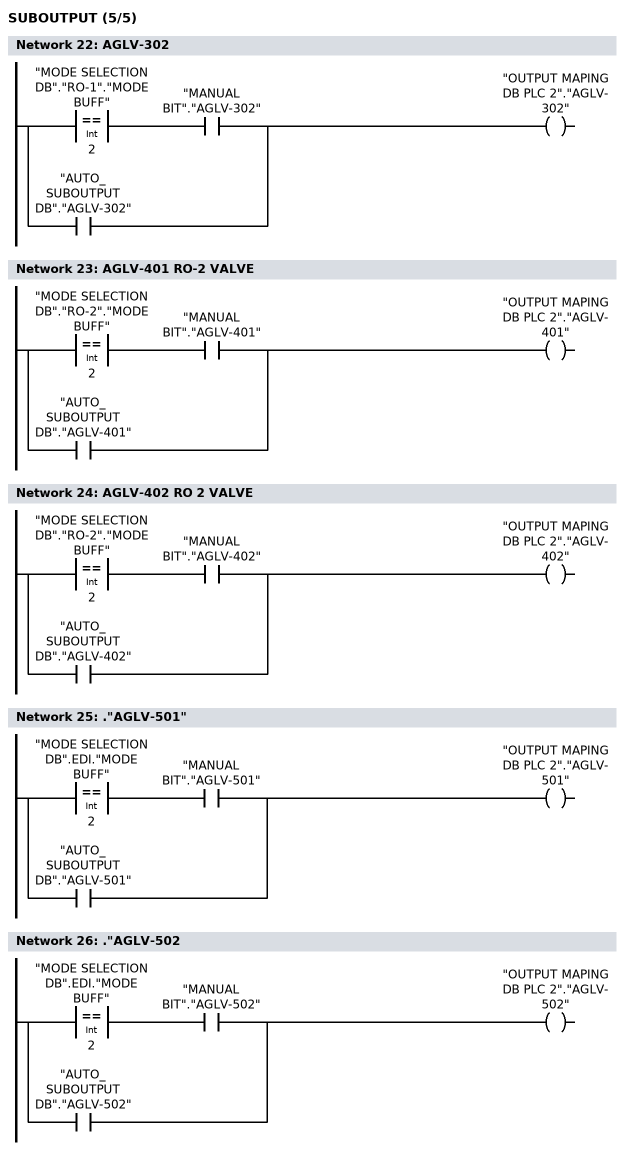
   RUNG wire#powerrail
      { S7_Templates := "SrcType := Int" } EQ_Contact(in1 := "MODE SELECTION DB"."RO-1"."MODE BUFF", in2 := 2)
      Contact( "MANUAL BIT"."AGLV-302" )
      wire#w1
      Coil( "OUTPUT MAPING DB PLC 2"."AGLV-302" )
   END_RUNG
   RUNG wire#powerrail
      Contact( "AUTO_SUBOUTPUT DB"."AGLV-302" )
   END_RUNG wire#w1
   // the same network as SCL:
   "OUTPUT MAPING DB PLC 2"."AGLV-302" := (("MODE SELECTION DB"."RO-1"."MODE BUFF" = 2) AND "MANUAL BIT"."AGLV-302") OR "AUTO_SUBOUTPUT DB"."AGLV-302";
END_REGION

REGION Network 23: AGLV-401 RO-2 VALVE
   RUNG wire#powerrail
      { S7_Templates := "SrcType := Int" } EQ_Contact(in1 := "MODE SELECTION DB"."RO-2"."MODE BUFF", in2 := 2)
      Contact( "MANUAL BIT"."AGLV-401" )
      wire#w1
      Coil( "OUTPUT MAPING DB PLC 2"."AGLV-401" )
   END_RUNG
   RUNG wire#powerrail
      Contact( "AUTO_SUBOUTPUT DB"."AGLV-401" )
   END_RUNG wire#w1
   // the same network as SCL:
   "OUTPUT MAPING DB PLC 2"."AGLV-401" := (("MODE SELECTION DB"."RO-2"."MODE BUFF" = 2) AND "MANUAL BIT"."AGLV-401") OR "AUTO_SUBOUTPUT DB"."AGLV-401";
END_REGION

REGION Network 24: AGLV-402 RO 2 VALVE
   RUNG wire#powerrail
      { S7_Templates := "SrcType := Int" } EQ_Contact(in1 := "MODE SELECTION DB"."RO-2"."MODE BUFF", in2 := 2)
      Contact( "MANUAL BIT"."AGLV-402" )
      wire#w1
      Coil( "OUTPUT MAPING DB PLC 2"."AGLV-402" )
   END_RUNG
   RUNG wire#powerrail
      Contact( "AUTO_SUBOUTPUT DB"."AGLV-402" )
   END_RUNG wire#w1
   // the same network as SCL:
   "OUTPUT MAPING DB PLC 2"."AGLV-402" := (("MODE SELECTION DB"."RO-2"."MODE BUFF" = 2) AND "MANUAL BIT"."AGLV-402") OR "AUTO_SUBOUTPUT DB"."AGLV-402";
END_REGION

REGION Network 25: ."AGLV-501"
   RUNG wire#powerrail
      { S7_Templates := "SrcType := Int" } EQ_Contact(in1 := "MODE SELECTION DB".EDI."MODE BUFF", in2 := 2)
      Contact( "MANUAL BIT"."AGLV-501" )
      wire#w1
      Coil( "OUTPUT MAPING DB PLC 2"."AGLV-501" )
   END_RUNG
   RUNG wire#powerrail
      Contact( "AUTO_SUBOUTPUT DB"."AGLV-501" )
   END_RUNG wire#w1
   // the same network as SCL:
   "OUTPUT MAPING DB PLC 2"."AGLV-501" := (("MODE SELECTION DB".EDI."MODE BUFF" = 2) AND "MANUAL BIT"."AGLV-501") OR "AUTO_SUBOUTPUT DB"."AGLV-501";
END_REGION

REGION Network 26: ."AGLV-502
   RUNG wire#powerrail
      { S7_Templates := "SrcType := Int" } EQ_Contact(in1 := "MODE SELECTION DB".EDI."MODE BUFF", in2 := 2)
      Contact( "MANUAL BIT"."AGLV-502" )
      wire#w1
      Coil( "OUTPUT MAPING DB PLC 2"."AGLV-502" )
   END_RUNG
   RUNG wire#powerrail
      Contact( "AUTO_SUBOUTPUT DB"."AGLV-502" )
   END_RUNG wire#w1
   // the same network as SCL:
   "OUTPUT MAPING DB PLC 2"."AGLV-502" := (("MODE SELECTION DB".EDI."MODE BUFF" = 2) AND "MANUAL BIT"."AGLV-502") OR "AUTO_SUBOUTPUT DB"."AGLV-502";
END_REGION
END_FUNCTION

FUNCTION "ALARM" : Void   // FC6, LAD
{ S7_Optimized_Access := 'TRUE' }
// stored: SetENOAutomatically false
   VAR_TEMP
      QQ : Bool;
   END_VAR
   VAR_TEMP   // added for the SCL form of the ladder/FBD networks
      _w1 : Bool;
   END_VAR
BEGIN

REGION Network 1: ALARM RESET (MASTER TO SLAVE)
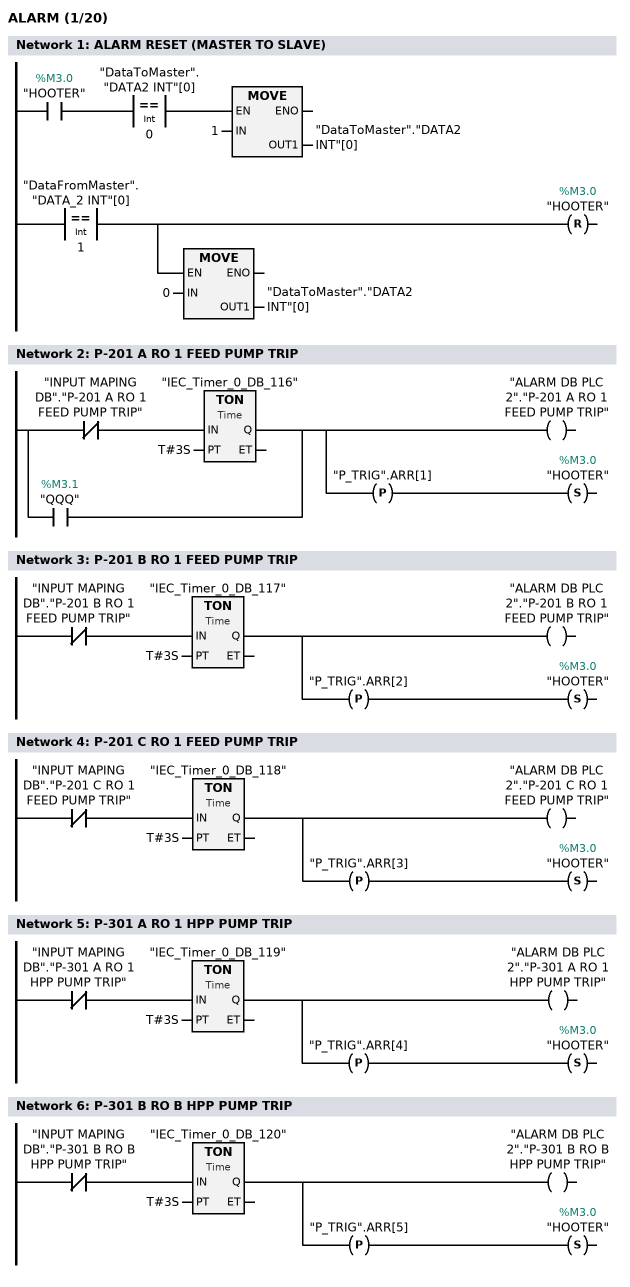
   RUNG wire#powerrail
      Contact( "HOOTER" )
      { S7_Templates := "SrcType := Int" } EQ_Contact(in1 := "DataToMaster"."DATA2 INT"[0], in2 := 0)
      Move(in := 1, out1 => "DataToMaster"."DATA2 INT"[0])
   END_RUNG
   RUNG wire#powerrail
      { S7_Templates := "SrcType := Int" } EQ_Contact(in1 := "DataFromMaster"."DATA_2 INT"[0], in2 := 1)
      wire#w1
      R_Coil( "HOOTER" )
   END_RUNG
   RUNG wire#w1
      Move(in := 0, out1 => "DataToMaster"."DATA2 INT"[0])
   END_RUNG
   // the same network as SCL:
   IF "HOOTER" AND ("DataToMaster"."DATA2 INT"[0] = 0) THEN "DataToMaster"."DATA2 INT"[0] := 1; END_IF;
   IF "DataFromMaster"."DATA_2 INT"[0] = 1 THEN
       "HOOTER" := FALSE;
       "DataToMaster"."DATA2 INT"[0] := 0;
   END_IF;
END_REGION

REGION Network 2: P-201 A RO 1 FEED PUMP TRIP
   RUNG wire#powerrail
      I_Contact( "INPUT MAPING DB"."P-201 A RO 1 FEED PUMP TRIP" )
      { S7_Templates := "time_type := Time" } "IEC_Timer_0_DB_116".TON(pt := T#3S, et =>)
      wire#w1
      Coil( "ALARM DB PLC 2"."P-201 A RO 1 FEED PUMP TRIP" )
   END_RUNG
   RUNG wire#powerrail
      Contact( "QQQ" )
   END_RUNG wire#w1
   RUNG wire#w1
      P_Trig( "P_TRIG".ARR[1] )
      S_Coil( "HOOTER" )
   END_RUNG
   // the same network as SCL:
   "IEC_Timer_0_DB_116".TON(IN := NOT "INPUT MAPING DB"."P-201 A RO 1 FEED PUMP TRIP", PT := T#3S);
   "ALARM DB PLC 2"."P-201 A RO 1 FEED PUMP TRIP" := "IEC_Timer_0_DB_116".Q OR "QQQ";
   #_w1 := "ALARM DB PLC 2"."P-201 A RO 1 FEED PUMP TRIP" AND NOT "P_TRIG".ARR[1];   // rising edge
   "P_TRIG".ARR[1] := "ALARM DB PLC 2"."P-201 A RO 1 FEED PUMP TRIP";
   IF #_w1 THEN "HOOTER" := TRUE; END_IF;
END_REGION

REGION Network 3: P-201 B RO 1 FEED PUMP TRIP
   RUNG wire#powerrail
      I_Contact( "INPUT MAPING DB"."P-201 B RO 1 FEED PUMP TRIP" )
      { S7_Templates := "time_type := Time" } "IEC_Timer_0_DB_117".TON(pt := T#3S, et =>)
      wire#w1
      Coil( "ALARM DB PLC 2"."P-201 B RO 1 FEED PUMP TRIP" )
   END_RUNG
   RUNG wire#w1
      P_Trig( "P_TRIG".ARR[2] )
      S_Coil( "HOOTER" )
   END_RUNG
   // the same network as SCL:
   "IEC_Timer_0_DB_117".TON(IN := NOT "INPUT MAPING DB"."P-201 B RO 1 FEED PUMP TRIP", PT := T#3S);
   "ALARM DB PLC 2"."P-201 B RO 1 FEED PUMP TRIP" := "IEC_Timer_0_DB_117".Q;
   #_w1 := "IEC_Timer_0_DB_117".Q AND NOT "P_TRIG".ARR[2];   // rising edge
   "P_TRIG".ARR[2] := "IEC_Timer_0_DB_117".Q;
   IF #_w1 THEN "HOOTER" := TRUE; END_IF;
END_REGION

REGION Network 4: P-201 C RO 1 FEED PUMP TRIP
   RUNG wire#powerrail
      I_Contact( "INPUT MAPING DB"."P-201 C RO 1 FEED PUMP TRIP" )
      { S7_Templates := "time_type := Time" } "IEC_Timer_0_DB_118".TON(pt := T#3S, et =>)
      wire#w1
      Coil( "ALARM DB PLC 2"."P-201 C RO 1 FEED PUMP TRIP" )
   END_RUNG
   RUNG wire#w1
      P_Trig( "P_TRIG".ARR[3] )
      S_Coil( "HOOTER" )
   END_RUNG
   // the same network as SCL:
   "IEC_Timer_0_DB_118".TON(IN := NOT "INPUT MAPING DB"."P-201 C RO 1 FEED PUMP TRIP", PT := T#3S);
   "ALARM DB PLC 2"."P-201 C RO 1 FEED PUMP TRIP" := "IEC_Timer_0_DB_118".Q;
   #_w1 := "IEC_Timer_0_DB_118".Q AND NOT "P_TRIG".ARR[3];   // rising edge
   "P_TRIG".ARR[3] := "IEC_Timer_0_DB_118".Q;
   IF #_w1 THEN "HOOTER" := TRUE; END_IF;
END_REGION

REGION Network 5: P-301 A RO 1 HPP PUMP TRIP
   RUNG wire#powerrail
      I_Contact( "INPUT MAPING DB"."P-301 A RO 1 HPP PUMP TRIP" )
      { S7_Templates := "time_type := Time" } "IEC_Timer_0_DB_119".TON(pt := T#3S, et =>)
      wire#w1
      Coil( "ALARM DB PLC 2"."P-301 A RO 1 HPP PUMP TRIP" )
   END_RUNG
   RUNG wire#w1
      P_Trig( "P_TRIG".ARR[4] )
      S_Coil( "HOOTER" )
   END_RUNG
   // the same network as SCL:
   "IEC_Timer_0_DB_119".TON(IN := NOT "INPUT MAPING DB"."P-301 A RO 1 HPP PUMP TRIP", PT := T#3S);
   "ALARM DB PLC 2"."P-301 A RO 1 HPP PUMP TRIP" := "IEC_Timer_0_DB_119".Q;
   #_w1 := "IEC_Timer_0_DB_119".Q AND NOT "P_TRIG".ARR[4];   // rising edge
   "P_TRIG".ARR[4] := "IEC_Timer_0_DB_119".Q;
   IF #_w1 THEN "HOOTER" := TRUE; END_IF;
END_REGION

REGION Network 6: P-301 B RO B HPP PUMP TRIP
   RUNG wire#powerrail
      I_Contact( "INPUT MAPING DB"."P-301 B RO B HPP PUMP TRIP" )
      { S7_Templates := "time_type := Time" } "IEC_Timer_0_DB_120".TON(pt := T#3S, et =>)
      wire#w1
      Coil( "ALARM DB PLC 2"."P-301 B RO B HPP PUMP TRIP" )
   END_RUNG
   RUNG wire#w1
      P_Trig( "P_TRIG".ARR[5] )
      S_Coil( "HOOTER" )
   END_RUNG
   // the same network as SCL:
   "IEC_Timer_0_DB_120".TON(IN := NOT "INPUT MAPING DB"."P-301 B RO B HPP PUMP TRIP", PT := T#3S);
   "ALARM DB PLC 2"."P-301 B RO B HPP PUMP TRIP" := "IEC_Timer_0_DB_120".Q;
   #_w1 := "IEC_Timer_0_DB_120".Q AND NOT "P_TRIG".ARR[5];   // rising edge
   "P_TRIG".ARR[5] := "IEC_Timer_0_DB_120".Q;
   IF #_w1 THEN "HOOTER" := TRUE; END_IF;
END_REGION

REGION Network 7: P-401 A RO 2 FEED PUMP TRIP
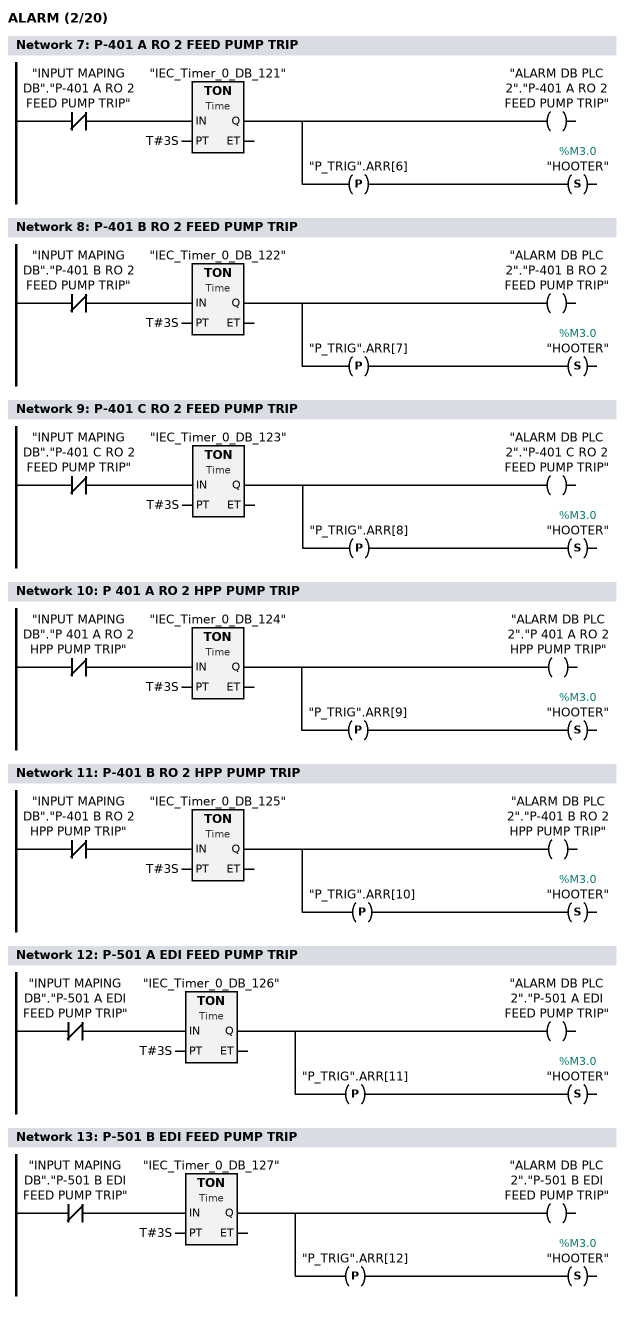
   RUNG wire#powerrail
      I_Contact( "INPUT MAPING DB"."P-401 A RO 2 FEED PUMP TRIP" )
      { S7_Templates := "time_type := Time" } "IEC_Timer_0_DB_121".TON(pt := T#3S, et =>)
      wire#w1
      Coil( "ALARM DB PLC 2"."P-401 A RO 2 FEED PUMP TRIP" )
   END_RUNG
   RUNG wire#w1
      P_Trig( "P_TRIG".ARR[6] )
      S_Coil( "HOOTER" )
   END_RUNG
   // the same network as SCL:
   "IEC_Timer_0_DB_121".TON(IN := NOT "INPUT MAPING DB"."P-401 A RO 2 FEED PUMP TRIP", PT := T#3S);
   "ALARM DB PLC 2"."P-401 A RO 2 FEED PUMP TRIP" := "IEC_Timer_0_DB_121".Q;
   #_w1 := "IEC_Timer_0_DB_121".Q AND NOT "P_TRIG".ARR[6];   // rising edge
   "P_TRIG".ARR[6] := "IEC_Timer_0_DB_121".Q;
   IF #_w1 THEN "HOOTER" := TRUE; END_IF;
END_REGION

REGION Network 8: P-401 B RO 2 FEED PUMP TRIP
   RUNG wire#powerrail
      I_Contact( "INPUT MAPING DB"."P-401 B RO 2 FEED PUMP TRIP" )
      { S7_Templates := "time_type := Time" } "IEC_Timer_0_DB_122".TON(pt := T#3S, et =>)
      wire#w1
      Coil( "ALARM DB PLC 2"."P-401 B RO 2 FEED PUMP TRIP" )
   END_RUNG
   RUNG wire#w1
      P_Trig( "P_TRIG".ARR[7] )
      S_Coil( "HOOTER" )
   END_RUNG
   // the same network as SCL:
   "IEC_Timer_0_DB_122".TON(IN := NOT "INPUT MAPING DB"."P-401 B RO 2 FEED PUMP TRIP", PT := T#3S);
   "ALARM DB PLC 2"."P-401 B RO 2 FEED PUMP TRIP" := "IEC_Timer_0_DB_122".Q;
   #_w1 := "IEC_Timer_0_DB_122".Q AND NOT "P_TRIG".ARR[7];   // rising edge
   "P_TRIG".ARR[7] := "IEC_Timer_0_DB_122".Q;
   IF #_w1 THEN "HOOTER" := TRUE; END_IF;
END_REGION

REGION Network 9: P-401 C RO 2 FEED PUMP TRIP
   RUNG wire#powerrail
      I_Contact( "INPUT MAPING DB"."P-401 C RO 2 FEED PUMP TRIP" )
      { S7_Templates := "time_type := Time" } "IEC_Timer_0_DB_123".TON(pt := T#3S, et =>)
      wire#w1
      Coil( "ALARM DB PLC 2"."P-401 C RO 2 FEED PUMP TRIP" )
   END_RUNG
   RUNG wire#w1
      P_Trig( "P_TRIG".ARR[8] )
      S_Coil( "HOOTER" )
   END_RUNG
   // the same network as SCL:
   "IEC_Timer_0_DB_123".TON(IN := NOT "INPUT MAPING DB"."P-401 C RO 2 FEED PUMP TRIP", PT := T#3S);
   "ALARM DB PLC 2"."P-401 C RO 2 FEED PUMP TRIP" := "IEC_Timer_0_DB_123".Q;
   #_w1 := "IEC_Timer_0_DB_123".Q AND NOT "P_TRIG".ARR[8];   // rising edge
   "P_TRIG".ARR[8] := "IEC_Timer_0_DB_123".Q;
   IF #_w1 THEN "HOOTER" := TRUE; END_IF;
END_REGION

REGION Network 10: P 401 A RO 2 HPP PUMP TRIP
   RUNG wire#powerrail
      I_Contact( "INPUT MAPING DB"."P 401 A RO 2 HPP PUMP TRIP" )
      { S7_Templates := "time_type := Time" } "IEC_Timer_0_DB_124".TON(pt := T#3S, et =>)
      wire#w1
      Coil( "ALARM DB PLC 2"."P 401 A RO 2 HPP PUMP TRIP" )
   END_RUNG
   RUNG wire#w1
      P_Trig( "P_TRIG".ARR[9] )
      S_Coil( "HOOTER" )
   END_RUNG
   // the same network as SCL:
   "IEC_Timer_0_DB_124".TON(IN := NOT "INPUT MAPING DB"."P 401 A RO 2 HPP PUMP TRIP", PT := T#3S);
   "ALARM DB PLC 2"."P 401 A RO 2 HPP PUMP TRIP" := "IEC_Timer_0_DB_124".Q;
   #_w1 := "IEC_Timer_0_DB_124".Q AND NOT "P_TRIG".ARR[9];   // rising edge
   "P_TRIG".ARR[9] := "IEC_Timer_0_DB_124".Q;
   IF #_w1 THEN "HOOTER" := TRUE; END_IF;
END_REGION

REGION Network 11: P-401 B RO 2 HPP PUMP TRIP
   RUNG wire#powerrail
      I_Contact( "INPUT MAPING DB"."P-401 B RO 2 HPP PUMP TRIP" )
      { S7_Templates := "time_type := Time" } "IEC_Timer_0_DB_125".TON(pt := T#3S, et =>)
      wire#w1
      Coil( "ALARM DB PLC 2"."P-401 B RO 2 HPP PUMP TRIP" )
   END_RUNG
   RUNG wire#w1
      P_Trig( "P_TRIG".ARR[10] )
      S_Coil( "HOOTER" )
   END_RUNG
   // the same network as SCL:
   "IEC_Timer_0_DB_125".TON(IN := NOT "INPUT MAPING DB"."P-401 B RO 2 HPP PUMP TRIP", PT := T#3S);
   "ALARM DB PLC 2"."P-401 B RO 2 HPP PUMP TRIP" := "IEC_Timer_0_DB_125".Q;
   #_w1 := "IEC_Timer_0_DB_125".Q AND NOT "P_TRIG".ARR[10];   // rising edge
   "P_TRIG".ARR[10] := "IEC_Timer_0_DB_125".Q;
   IF #_w1 THEN "HOOTER" := TRUE; END_IF;
END_REGION

REGION Network 12: P-501 A EDI FEED PUMP TRIP
   RUNG wire#powerrail
      I_Contact( "INPUT MAPING DB"."P-501 A EDI FEED PUMP TRIP" )
      { S7_Templates := "time_type := Time" } "IEC_Timer_0_DB_126".TON(pt := T#3S, et =>)
      wire#w1
      Coil( "ALARM DB PLC 2"."P-501 A EDI FEED PUMP TRIP" )
   END_RUNG
   RUNG wire#w1
      P_Trig( "P_TRIG".ARR[11] )
      S_Coil( "HOOTER" )
   END_RUNG
   // the same network as SCL:
   "IEC_Timer_0_DB_126".TON(IN := NOT "INPUT MAPING DB"."P-501 A EDI FEED PUMP TRIP", PT := T#3S);
   "ALARM DB PLC 2"."P-501 A EDI FEED PUMP TRIP" := "IEC_Timer_0_DB_126".Q;
   #_w1 := "IEC_Timer_0_DB_126".Q AND NOT "P_TRIG".ARR[11];   // rising edge
   "P_TRIG".ARR[11] := "IEC_Timer_0_DB_126".Q;
   IF #_w1 THEN "HOOTER" := TRUE; END_IF;
END_REGION

REGION Network 13: P-501 B EDI FEED PUMP TRIP
   RUNG wire#powerrail
      I_Contact( "INPUT MAPING DB"."P-501 B EDI FEED PUMP TRIP" )
      { S7_Templates := "time_type := Time" } "IEC_Timer_0_DB_127".TON(pt := T#3S, et =>)
      wire#w1
      Coil( "ALARM DB PLC 2"."P-501 B EDI FEED PUMP TRIP" )
   END_RUNG
   RUNG wire#w1
      P_Trig( "P_TRIG".ARR[12] )
      S_Coil( "HOOTER" )
   END_RUNG
   // the same network as SCL:
   "IEC_Timer_0_DB_127".TON(IN := NOT "INPUT MAPING DB"."P-501 B EDI FEED PUMP TRIP", PT := T#3S);
   "ALARM DB PLC 2"."P-501 B EDI FEED PUMP TRIP" := "IEC_Timer_0_DB_127".Q;
   #_w1 := "IEC_Timer_0_DB_127".Q AND NOT "P_TRIG".ARR[12];   // rising edge
   "P_TRIG".ARR[12] := "IEC_Timer_0_DB_127".Q;
   IF #_w1 THEN "HOOTER" := TRUE; END_IF;
END_REGION

REGION Network 14: P-501 C EDI FEED PUMP TRIP
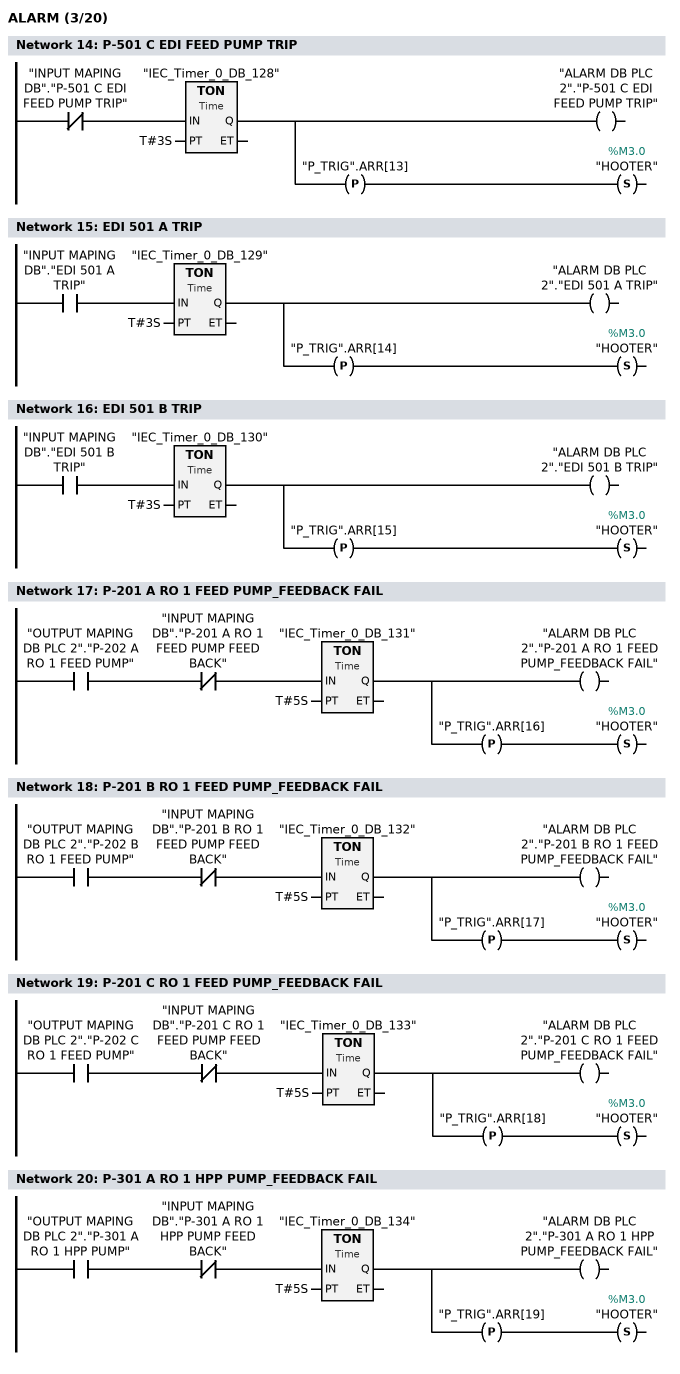
   RUNG wire#powerrail
      I_Contact( "INPUT MAPING DB"."P-501 C EDI FEED PUMP TRIP" )
      { S7_Templates := "time_type := Time" } "IEC_Timer_0_DB_128".TON(pt := T#3S, et =>)
      wire#w1
      Coil( "ALARM DB PLC 2"."P-501 C EDI FEED PUMP TRIP" )
   END_RUNG
   RUNG wire#w1
      P_Trig( "P_TRIG".ARR[13] )
      S_Coil( "HOOTER" )
   END_RUNG
   // the same network as SCL:
   "IEC_Timer_0_DB_128".TON(IN := NOT "INPUT MAPING DB"."P-501 C EDI FEED PUMP TRIP", PT := T#3S);
   "ALARM DB PLC 2"."P-501 C EDI FEED PUMP TRIP" := "IEC_Timer_0_DB_128".Q;
   #_w1 := "IEC_Timer_0_DB_128".Q AND NOT "P_TRIG".ARR[13];   // rising edge
   "P_TRIG".ARR[13] := "IEC_Timer_0_DB_128".Q;
   IF #_w1 THEN "HOOTER" := TRUE; END_IF;
END_REGION

REGION Network 15: EDI 501 A TRIP
   RUNG wire#powerrail
      Contact( "INPUT MAPING DB"."EDI 501 A TRIP" )
      { S7_Templates := "time_type := Time" } "IEC_Timer_0_DB_129".TON(pt := T#3S, et =>)
      wire#w1
      Coil( "ALARM DB PLC 2"."EDI 501 A TRIP" )
   END_RUNG
   RUNG wire#w1
      P_Trig( "P_TRIG".ARR[14] )
      S_Coil( "HOOTER" )
   END_RUNG
   // the same network as SCL:
   "IEC_Timer_0_DB_129".TON(IN := "INPUT MAPING DB"."EDI 501 A TRIP", PT := T#3S);
   "ALARM DB PLC 2"."EDI 501 A TRIP" := "IEC_Timer_0_DB_129".Q;
   #_w1 := "IEC_Timer_0_DB_129".Q AND NOT "P_TRIG".ARR[14];   // rising edge
   "P_TRIG".ARR[14] := "IEC_Timer_0_DB_129".Q;
   IF #_w1 THEN "HOOTER" := TRUE; END_IF;
END_REGION

REGION Network 16: EDI 501 B TRIP
   RUNG wire#powerrail
      Contact( "INPUT MAPING DB"."EDI 501 B TRIP" )
      { S7_Templates := "time_type := Time" } "IEC_Timer_0_DB_130".TON(pt := T#3S, et =>)
      wire#w1
      Coil( "ALARM DB PLC 2"."EDI 501 B TRIP" )
   END_RUNG
   RUNG wire#w1
      P_Trig( "P_TRIG".ARR[15] )
      S_Coil( "HOOTER" )
   END_RUNG
   // the same network as SCL:
   "IEC_Timer_0_DB_130".TON(IN := "INPUT MAPING DB"."EDI 501 B TRIP", PT := T#3S);
   "ALARM DB PLC 2"."EDI 501 B TRIP" := "IEC_Timer_0_DB_130".Q;
   #_w1 := "IEC_Timer_0_DB_130".Q AND NOT "P_TRIG".ARR[15];   // rising edge
   "P_TRIG".ARR[15] := "IEC_Timer_0_DB_130".Q;
   IF #_w1 THEN "HOOTER" := TRUE; END_IF;
END_REGION

REGION Network 17: P-201 A RO 1 FEED PUMP_FEEDBACK FAIL
   RUNG wire#powerrail
      Contact( "OUTPUT MAPING DB PLC 2"."P-202 A RO 1 FEED PUMP" )
      I_Contact( "INPUT MAPING DB"."P-201 A RO 1 FEED PUMP FEED BACK" )
      { S7_Templates := "time_type := Time" } "IEC_Timer_0_DB_131".TON(pt := T#5S, et =>)
      wire#w1
      Coil( "ALARM DB PLC 2"."P-201 A RO 1 FEED PUMP_FEEDBACK FAIL" )
   END_RUNG
   RUNG wire#w1
      P_Trig( "P_TRIG".ARR[16] )
      S_Coil( "HOOTER" )
   END_RUNG
   // the same network as SCL:
   "IEC_Timer_0_DB_131".TON(IN := "OUTPUT MAPING DB PLC 2"."P-202 A RO 1 FEED PUMP" AND NOT "INPUT MAPING DB"."P-201 A RO 1 FEED PUMP FEED BACK",
                           PT := T#5S);
   "ALARM DB PLC 2"."P-201 A RO 1 FEED PUMP_FEEDBACK FAIL" := "IEC_Timer_0_DB_131".Q;
   #_w1 := "IEC_Timer_0_DB_131".Q AND NOT "P_TRIG".ARR[16];   // rising edge
   "P_TRIG".ARR[16] := "IEC_Timer_0_DB_131".Q;
   IF #_w1 THEN "HOOTER" := TRUE; END_IF;
END_REGION

REGION Network 18: P-201 B RO 1 FEED PUMP_FEEDBACK FAIL
   RUNG wire#powerrail
      Contact( "OUTPUT MAPING DB PLC 2"."P-202 B RO 1 FEED PUMP" )
      I_Contact( "INPUT MAPING DB"."P-201 B RO 1 FEED PUMP FEED BACK" )
      { S7_Templates := "time_type := Time" } "IEC_Timer_0_DB_132".TON(pt := T#5S, et =>)
      wire#w1
      Coil( "ALARM DB PLC 2"."P-201 B RO 1 FEED PUMP_FEEDBACK FAIL" )
   END_RUNG
   RUNG wire#w1
      P_Trig( "P_TRIG".ARR[17] )
      S_Coil( "HOOTER" )
   END_RUNG
   // the same network as SCL:
   "IEC_Timer_0_DB_132".TON(IN := "OUTPUT MAPING DB PLC 2"."P-202 B RO 1 FEED PUMP" AND NOT "INPUT MAPING DB"."P-201 B RO 1 FEED PUMP FEED BACK",
                           PT := T#5S);
   "ALARM DB PLC 2"."P-201 B RO 1 FEED PUMP_FEEDBACK FAIL" := "IEC_Timer_0_DB_132".Q;
   #_w1 := "IEC_Timer_0_DB_132".Q AND NOT "P_TRIG".ARR[17];   // rising edge
   "P_TRIG".ARR[17] := "IEC_Timer_0_DB_132".Q;
   IF #_w1 THEN "HOOTER" := TRUE; END_IF;
END_REGION

REGION Network 19: P-201 C RO 1 FEED PUMP_FEEDBACK FAIL
   RUNG wire#powerrail
      Contact( "OUTPUT MAPING DB PLC 2"."P-202 C RO 1 FEED PUMP" )
      I_Contact( "INPUT MAPING DB"."P-201 C RO 1 FEED PUMP FEED BACK" )
      { S7_Templates := "time_type := Time" } "IEC_Timer_0_DB_133".TON(pt := T#5S, et =>)
      wire#w1
      Coil( "ALARM DB PLC 2"."P-201 C RO 1 FEED PUMP_FEEDBACK FAIL" )
   END_RUNG
   RUNG wire#w1
      P_Trig( "P_TRIG".ARR[18] )
      S_Coil( "HOOTER" )
   END_RUNG
   // the same network as SCL:
   "IEC_Timer_0_DB_133".TON(IN := "OUTPUT MAPING DB PLC 2"."P-202 C RO 1 FEED PUMP" AND NOT "INPUT MAPING DB"."P-201 C RO 1 FEED PUMP FEED BACK",
                           PT := T#5S);
   "ALARM DB PLC 2"."P-201 C RO 1 FEED PUMP_FEEDBACK FAIL" := "IEC_Timer_0_DB_133".Q;
   #_w1 := "IEC_Timer_0_DB_133".Q AND NOT "P_TRIG".ARR[18];   // rising edge
   "P_TRIG".ARR[18] := "IEC_Timer_0_DB_133".Q;
   IF #_w1 THEN "HOOTER" := TRUE; END_IF;
END_REGION

REGION Network 20: P-301 A RO 1 HPP PUMP_FEEDBACK FAIL
   RUNG wire#powerrail
      Contact( "OUTPUT MAPING DB PLC 2"."P-301 A RO 1 HPP PUMP" )
      I_Contact( "INPUT MAPING DB"."P-301 A RO 1 HPP PUMP FEED BACK" )
      { S7_Templates := "time_type := Time" } "IEC_Timer_0_DB_134".TON(pt := T#5S, et =>)
      wire#w1
      Coil( "ALARM DB PLC 2"."P-301 A RO 1 HPP PUMP_FEEDBACK FAIL" )
   END_RUNG
   RUNG wire#w1
      P_Trig( "P_TRIG".ARR[19] )
      S_Coil( "HOOTER" )
   END_RUNG
   // the same network as SCL:
   "IEC_Timer_0_DB_134".TON(IN := "OUTPUT MAPING DB PLC 2"."P-301 A RO 1 HPP PUMP" AND NOT "INPUT MAPING DB"."P-301 A RO 1 HPP PUMP FEED BACK",
                           PT := T#5S);
   "ALARM DB PLC 2"."P-301 A RO 1 HPP PUMP_FEEDBACK FAIL" := "IEC_Timer_0_DB_134".Q;
   #_w1 := "IEC_Timer_0_DB_134".Q AND NOT "P_TRIG".ARR[19];   // rising edge
   "P_TRIG".ARR[19] := "IEC_Timer_0_DB_134".Q;
   IF #_w1 THEN "HOOTER" := TRUE; END_IF;
END_REGION

REGION Network 21: P-301 B RO B HPP PUMP_FEEDBACK FAIL
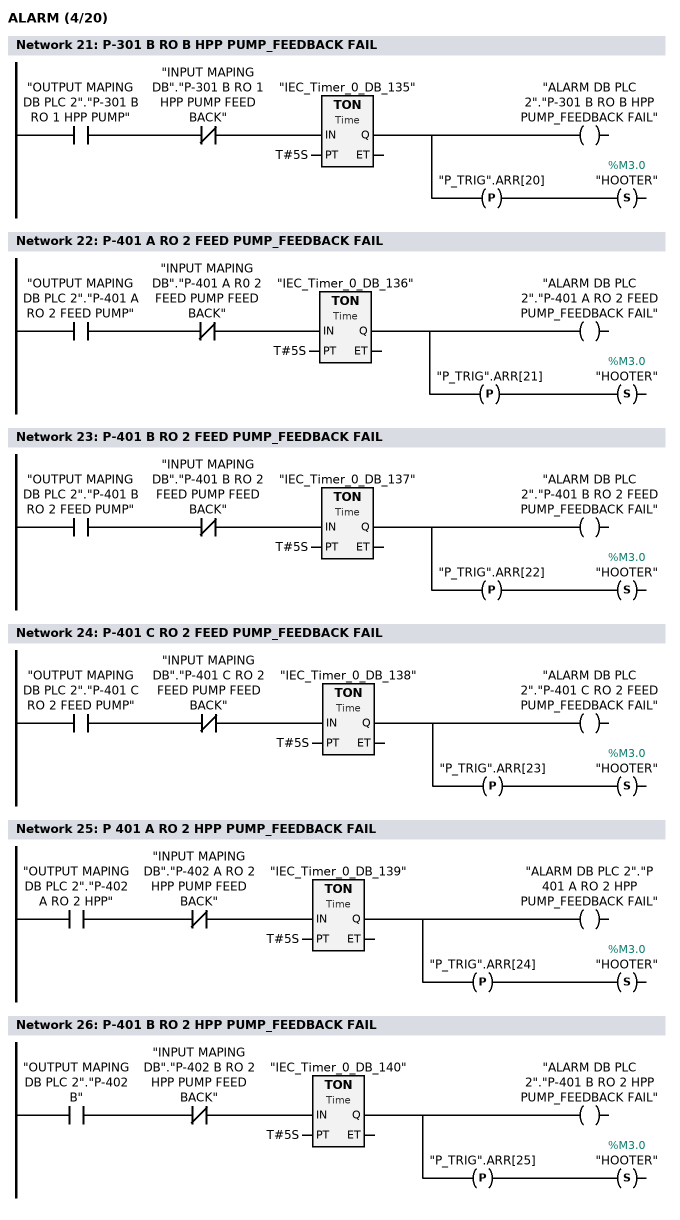
   RUNG wire#powerrail
      Contact( "OUTPUT MAPING DB PLC 2"."P-301 B RO 1 HPP PUMP" )
      I_Contact( "INPUT MAPING DB"."P-301 B RO 1 HPP PUMP FEED BACK" )
      { S7_Templates := "time_type := Time" } "IEC_Timer_0_DB_135".TON(pt := T#5S, et =>)
      wire#w1
      Coil( "ALARM DB PLC 2"."P-301 B RO B HPP PUMP_FEEDBACK FAIL" )
   END_RUNG
   RUNG wire#w1
      P_Trig( "P_TRIG".ARR[20] )
      S_Coil( "HOOTER" )
   END_RUNG
   // the same network as SCL:
   "IEC_Timer_0_DB_135".TON(IN := "OUTPUT MAPING DB PLC 2"."P-301 B RO 1 HPP PUMP" AND NOT "INPUT MAPING DB"."P-301 B RO 1 HPP PUMP FEED BACK",
                           PT := T#5S);
   "ALARM DB PLC 2"."P-301 B RO B HPP PUMP_FEEDBACK FAIL" := "IEC_Timer_0_DB_135".Q;
   #_w1 := "IEC_Timer_0_DB_135".Q AND NOT "P_TRIG".ARR[20];   // rising edge
   "P_TRIG".ARR[20] := "IEC_Timer_0_DB_135".Q;
   IF #_w1 THEN "HOOTER" := TRUE; END_IF;
END_REGION

REGION Network 22: P-401 A RO 2 FEED PUMP_FEEDBACK FAIL
   RUNG wire#powerrail
      Contact( "OUTPUT MAPING DB PLC 2"."P-401 A RO 2 FEED PUMP" )
      I_Contact( "INPUT MAPING DB"."P-401 A R0 2 FEED PUMP FEED BACK" )
      { S7_Templates := "time_type := Time" } "IEC_Timer_0_DB_136".TON(pt := T#5S, et =>)
      wire#w1
      Coil( "ALARM DB PLC 2"."P-401 A RO 2 FEED PUMP_FEEDBACK FAIL" )
   END_RUNG
   RUNG wire#w1
      P_Trig( "P_TRIG".ARR[21] )
      S_Coil( "HOOTER" )
   END_RUNG
   // the same network as SCL:
   "IEC_Timer_0_DB_136".TON(IN := "OUTPUT MAPING DB PLC 2"."P-401 A RO 2 FEED PUMP" AND NOT "INPUT MAPING DB"."P-401 A R0 2 FEED PUMP FEED BACK",
                           PT := T#5S);
   "ALARM DB PLC 2"."P-401 A RO 2 FEED PUMP_FEEDBACK FAIL" := "IEC_Timer_0_DB_136".Q;
   #_w1 := "IEC_Timer_0_DB_136".Q AND NOT "P_TRIG".ARR[21];   // rising edge
   "P_TRIG".ARR[21] := "IEC_Timer_0_DB_136".Q;
   IF #_w1 THEN "HOOTER" := TRUE; END_IF;
END_REGION

REGION Network 23: P-401 B RO 2 FEED PUMP_FEEDBACK FAIL
   RUNG wire#powerrail
      Contact( "OUTPUT MAPING DB PLC 2"."P-401 B RO 2 FEED PUMP" )
      I_Contact( "INPUT MAPING DB"."P-401 B RO 2 FEED PUMP FEED BACK" )
      { S7_Templates := "time_type := Time" } "IEC_Timer_0_DB_137".TON(pt := T#5S, et =>)
      wire#w1
      Coil( "ALARM DB PLC 2"."P-401 B RO 2 FEED PUMP_FEEDBACK FAIL" )
   END_RUNG
   RUNG wire#w1
      P_Trig( "P_TRIG".ARR[22] )
      S_Coil( "HOOTER" )
   END_RUNG
   // the same network as SCL:
   "IEC_Timer_0_DB_137".TON(IN := "OUTPUT MAPING DB PLC 2"."P-401 B RO 2 FEED PUMP" AND NOT "INPUT MAPING DB"."P-401 B RO 2 FEED PUMP FEED BACK",
                           PT := T#5S);
   "ALARM DB PLC 2"."P-401 B RO 2 FEED PUMP_FEEDBACK FAIL" := "IEC_Timer_0_DB_137".Q;
   #_w1 := "IEC_Timer_0_DB_137".Q AND NOT "P_TRIG".ARR[22];   // rising edge
   "P_TRIG".ARR[22] := "IEC_Timer_0_DB_137".Q;
   IF #_w1 THEN "HOOTER" := TRUE; END_IF;
END_REGION

REGION Network 24: P-401 C RO 2 FEED PUMP_FEEDBACK FAIL
   RUNG wire#powerrail
      Contact( "OUTPUT MAPING DB PLC 2"."P-401 C RO 2 FEED PUMP" )
      I_Contact( "INPUT MAPING DB"."P-401 C RO 2 FEED PUMP FEED BACK" )
      { S7_Templates := "time_type := Time" } "IEC_Timer_0_DB_138".TON(pt := T#5S, et =>)
      wire#w1
      Coil( "ALARM DB PLC 2"."P-401 C RO 2 FEED PUMP_FEEDBACK FAIL" )
   END_RUNG
   RUNG wire#w1
      P_Trig( "P_TRIG".ARR[23] )
      S_Coil( "HOOTER" )
   END_RUNG
   // the same network as SCL:
   "IEC_Timer_0_DB_138".TON(IN := "OUTPUT MAPING DB PLC 2"."P-401 C RO 2 FEED PUMP" AND NOT "INPUT MAPING DB"."P-401 C RO 2 FEED PUMP FEED BACK",
                           PT := T#5S);
   "ALARM DB PLC 2"."P-401 C RO 2 FEED PUMP_FEEDBACK FAIL" := "IEC_Timer_0_DB_138".Q;
   #_w1 := "IEC_Timer_0_DB_138".Q AND NOT "P_TRIG".ARR[23];   // rising edge
   "P_TRIG".ARR[23] := "IEC_Timer_0_DB_138".Q;
   IF #_w1 THEN "HOOTER" := TRUE; END_IF;
END_REGION

REGION Network 25: P 401 A RO 2 HPP PUMP_FEEDBACK FAIL
   RUNG wire#powerrail
      Contact( "OUTPUT MAPING DB PLC 2"."P-402  A RO 2 HPP" )
      I_Contact( "INPUT MAPING DB"."P-402 A RO 2 HPP PUMP FEED BACK" )
      { S7_Templates := "time_type := Time" } "IEC_Timer_0_DB_139".TON(pt := T#5S, et =>)
      wire#w1
      Coil( "ALARM DB PLC 2"."P 401 A RO 2 HPP PUMP_FEEDBACK FAIL" )
   END_RUNG
   RUNG wire#w1
      P_Trig( "P_TRIG".ARR[24] )
      S_Coil( "HOOTER" )
   END_RUNG
   // the same network as SCL:
   "IEC_Timer_0_DB_139".TON(IN := "OUTPUT MAPING DB PLC 2"."P-402  A RO 2 HPP" AND NOT "INPUT MAPING DB"."P-402 A RO 2 HPP PUMP FEED BACK",
                           PT := T#5S);
   "ALARM DB PLC 2"."P 401 A RO 2 HPP PUMP_FEEDBACK FAIL" := "IEC_Timer_0_DB_139".Q;
   #_w1 := "IEC_Timer_0_DB_139".Q AND NOT "P_TRIG".ARR[24];   // rising edge
   "P_TRIG".ARR[24] := "IEC_Timer_0_DB_139".Q;
   IF #_w1 THEN "HOOTER" := TRUE; END_IF;
END_REGION

REGION Network 26: P-401 B RO 2 HPP PUMP_FEEDBACK FAIL
   RUNG wire#powerrail
      Contact( "OUTPUT MAPING DB PLC 2"."P-402 B" )
      I_Contact( "INPUT MAPING DB"."P-402 B RO 2 HPP PUMP FEED BACK" )
      { S7_Templates := "time_type := Time" } "IEC_Timer_0_DB_140".TON(pt := T#5S, et =>)
      wire#w1
      Coil( "ALARM DB PLC 2"."P-401 B RO 2 HPP PUMP_FEEDBACK FAIL" )
   END_RUNG
   RUNG wire#w1
      P_Trig( "P_TRIG".ARR[25] )
      S_Coil( "HOOTER" )
   END_RUNG
   // the same network as SCL:
   "IEC_Timer_0_DB_140".TON(IN := "OUTPUT MAPING DB PLC 2"."P-402 B" AND NOT "INPUT MAPING DB"."P-402 B RO 2 HPP PUMP FEED BACK",
                           PT := T#5S);
   "ALARM DB PLC 2"."P-401 B RO 2 HPP PUMP_FEEDBACK FAIL" := "IEC_Timer_0_DB_140".Q;
   #_w1 := "IEC_Timer_0_DB_140".Q AND NOT "P_TRIG".ARR[25];   // rising edge
   "P_TRIG".ARR[25] := "IEC_Timer_0_DB_140".Q;
   IF #_w1 THEN "HOOTER" := TRUE; END_IF;
END_REGION

REGION Network 27: P-501 A EDI FEED PUMP_FEEDBACK FAIL
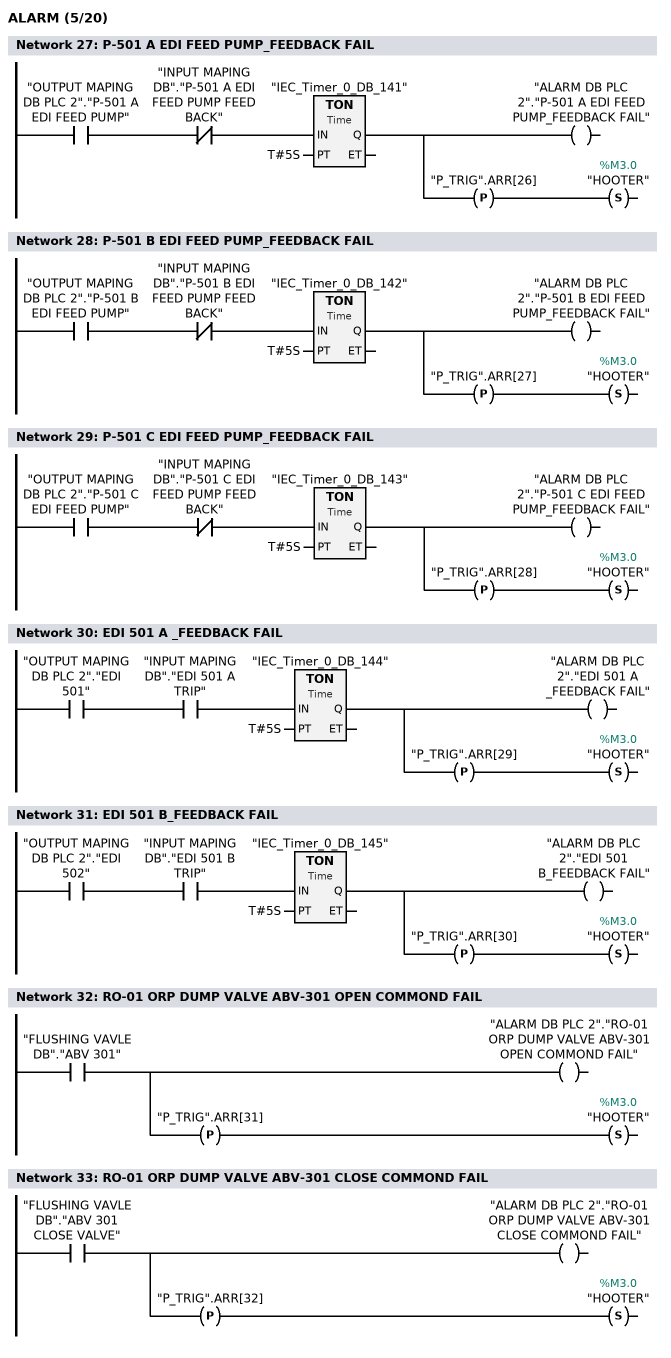
   RUNG wire#powerrail
      Contact( "OUTPUT MAPING DB PLC 2"."P-501 A EDI FEED PUMP" )
      I_Contact( "INPUT MAPING DB"."P-501 A EDI FEED PUMP FEED BACK" )
      { S7_Templates := "time_type := Time" } "IEC_Timer_0_DB_141".TON(pt := T#5S, et =>)
      wire#w1
      Coil( "ALARM DB PLC 2"."P-501 A EDI FEED PUMP_FEEDBACK FAIL" )
   END_RUNG
   RUNG wire#w1
      P_Trig( "P_TRIG".ARR[26] )
      S_Coil( "HOOTER" )
   END_RUNG
   // the same network as SCL:
   "IEC_Timer_0_DB_141".TON(IN := "OUTPUT MAPING DB PLC 2"."P-501 A EDI FEED PUMP" AND NOT "INPUT MAPING DB"."P-501 A EDI FEED PUMP FEED BACK",
                           PT := T#5S);
   "ALARM DB PLC 2"."P-501 A EDI FEED PUMP_FEEDBACK FAIL" := "IEC_Timer_0_DB_141".Q;
   #_w1 := "IEC_Timer_0_DB_141".Q AND NOT "P_TRIG".ARR[26];   // rising edge
   "P_TRIG".ARR[26] := "IEC_Timer_0_DB_141".Q;
   IF #_w1 THEN "HOOTER" := TRUE; END_IF;
END_REGION

REGION Network 28: P-501 B EDI FEED PUMP_FEEDBACK FAIL
   RUNG wire#powerrail
      Contact( "OUTPUT MAPING DB PLC 2"."P-501 B EDI FEED PUMP" )
      I_Contact( "INPUT MAPING DB"."P-501 B EDI FEED PUMP FEED BACK" )
      { S7_Templates := "time_type := Time" } "IEC_Timer_0_DB_142".TON(pt := T#5S, et =>)
      wire#w1
      Coil( "ALARM DB PLC 2"."P-501 B EDI FEED PUMP_FEEDBACK FAIL" )
   END_RUNG
   RUNG wire#w1
      P_Trig( "P_TRIG".ARR[27] )
      S_Coil( "HOOTER" )
   END_RUNG
   // the same network as SCL:
   "IEC_Timer_0_DB_142".TON(IN := "OUTPUT MAPING DB PLC 2"."P-501 B EDI FEED PUMP" AND NOT "INPUT MAPING DB"."P-501 B EDI FEED PUMP FEED BACK",
                           PT := T#5S);
   "ALARM DB PLC 2"."P-501 B EDI FEED PUMP_FEEDBACK FAIL" := "IEC_Timer_0_DB_142".Q;
   #_w1 := "IEC_Timer_0_DB_142".Q AND NOT "P_TRIG".ARR[27];   // rising edge
   "P_TRIG".ARR[27] := "IEC_Timer_0_DB_142".Q;
   IF #_w1 THEN "HOOTER" := TRUE; END_IF;
END_REGION

REGION Network 29: P-501 C EDI FEED PUMP_FEEDBACK FAIL
   RUNG wire#powerrail
      Contact( "OUTPUT MAPING DB PLC 2"."P-501 C EDI FEED PUMP" )
      I_Contact( "INPUT MAPING DB"."P-501 C EDI FEED PUMP FEED BACK" )
      { S7_Templates := "time_type := Time" } "IEC_Timer_0_DB_143".TON(pt := T#5S, et =>)
      wire#w1
      Coil( "ALARM DB PLC 2"."P-501 C EDI FEED PUMP_FEEDBACK FAIL" )
   END_RUNG
   RUNG wire#w1
      P_Trig( "P_TRIG".ARR[28] )
      S_Coil( "HOOTER" )
   END_RUNG
   // the same network as SCL:
   "IEC_Timer_0_DB_143".TON(IN := "OUTPUT MAPING DB PLC 2"."P-501 C EDI FEED PUMP" AND NOT "INPUT MAPING DB"."P-501 C EDI FEED PUMP FEED BACK",
                           PT := T#5S);
   "ALARM DB PLC 2"."P-501 C EDI FEED PUMP_FEEDBACK FAIL" := "IEC_Timer_0_DB_143".Q;
   #_w1 := "IEC_Timer_0_DB_143".Q AND NOT "P_TRIG".ARR[28];   // rising edge
   "P_TRIG".ARR[28] := "IEC_Timer_0_DB_143".Q;
   IF #_w1 THEN "HOOTER" := TRUE; END_IF;
END_REGION

REGION Network 30: EDI 501 A _FEEDBACK FAIL
   RUNG wire#powerrail
      Contact( "OUTPUT MAPING DB PLC 2"."EDI 501" )
      Contact( "INPUT MAPING DB"."EDI 501 A TRIP" )
      { S7_Templates := "time_type := Time" } "IEC_Timer_0_DB_144".TON(pt := T#5S, et =>)
      wire#w1
      Coil( "ALARM DB PLC 2"."EDI 501 A _FEEDBACK FAIL" )
   END_RUNG
   RUNG wire#w1
      P_Trig( "P_TRIG".ARR[29] )
      S_Coil( "HOOTER" )
   END_RUNG
   // the same network as SCL:
   "IEC_Timer_0_DB_144".TON(IN := "OUTPUT MAPING DB PLC 2"."EDI 501" AND "INPUT MAPING DB"."EDI 501 A TRIP",
                           PT := T#5S);
   "ALARM DB PLC 2"."EDI 501 A _FEEDBACK FAIL" := "IEC_Timer_0_DB_144".Q;
   #_w1 := "IEC_Timer_0_DB_144".Q AND NOT "P_TRIG".ARR[29];   // rising edge
   "P_TRIG".ARR[29] := "IEC_Timer_0_DB_144".Q;
   IF #_w1 THEN "HOOTER" := TRUE; END_IF;
END_REGION

REGION Network 31: EDI 501 B_FEEDBACK FAIL
   RUNG wire#powerrail
      Contact( "OUTPUT MAPING DB PLC 2"."EDI 502" )
      Contact( "INPUT MAPING DB"."EDI 501 B TRIP" )
      { S7_Templates := "time_type := Time" } "IEC_Timer_0_DB_145".TON(pt := T#5S, et =>)
      wire#w1
      Coil( "ALARM DB PLC 2"."EDI 501 B_FEEDBACK FAIL" )
   END_RUNG
   RUNG wire#w1
      P_Trig( "P_TRIG".ARR[30] )
      S_Coil( "HOOTER" )
   END_RUNG
   // the same network as SCL:
   "IEC_Timer_0_DB_145".TON(IN := "OUTPUT MAPING DB PLC 2"."EDI 502" AND "INPUT MAPING DB"."EDI 501 B TRIP",
                           PT := T#5S);
   "ALARM DB PLC 2"."EDI 501 B_FEEDBACK FAIL" := "IEC_Timer_0_DB_145".Q;
   #_w1 := "IEC_Timer_0_DB_145".Q AND NOT "P_TRIG".ARR[30];   // rising edge
   "P_TRIG".ARR[30] := "IEC_Timer_0_DB_145".Q;
   IF #_w1 THEN "HOOTER" := TRUE; END_IF;
END_REGION

REGION Network 32: RO-01 ORP DUMP VALVE ABV-301 OPEN COMMOND FAIL
   RUNG wire#powerrail
      Contact( "FLUSHING VAVLE DB"."ABV 301" )
      wire#w1
      Coil( "ALARM DB PLC 2"."RO-01 ORP DUMP VALVE ABV-301 OPEN COMMOND FAIL" )
   END_RUNG
   RUNG wire#w1
      P_Trig( "P_TRIG".ARR[31] )
      S_Coil( "HOOTER" )
   END_RUNG
   // the same network as SCL:
   "ALARM DB PLC 2"."RO-01 ORP DUMP VALVE ABV-301 OPEN COMMOND FAIL" := "FLUSHING VAVLE DB"."ABV 301";
   #_w1 := "FLUSHING VAVLE DB"."ABV 301" AND NOT "P_TRIG".ARR[31];   // rising edge
   "P_TRIG".ARR[31] := "FLUSHING VAVLE DB"."ABV 301";
   IF #_w1 THEN "HOOTER" := TRUE; END_IF;
END_REGION

REGION Network 33: RO-01 ORP DUMP VALVE ABV-301 CLOSE COMMOND FAIL
   RUNG wire#powerrail
      Contact( "FLUSHING VAVLE DB"."ABV 301 CLOSE VALVE" )
      wire#w1
      Coil( "ALARM DB PLC 2"."RO-01 ORP DUMP VALVE ABV-301 CLOSE COMMOND FAIL" )
   END_RUNG
   RUNG wire#w1
      P_Trig( "P_TRIG".ARR[32] )
      S_Coil( "HOOTER" )
   END_RUNG
   // the same network as SCL:
   "ALARM DB PLC 2"."RO-01 ORP DUMP VALVE ABV-301 CLOSE COMMOND FAIL" := "FLUSHING VAVLE DB"."ABV 301 CLOSE VALVE";
   #_w1 := "FLUSHING VAVLE DB"."ABV 301 CLOSE VALVE" AND NOT "P_TRIG".ARR[32];   // rising edge
   "P_TRIG".ARR[32] := "FLUSHING VAVLE DB"."ABV 301 CLOSE VALVE";
   IF #_w1 THEN "HOOTER" := TRUE; END_IF;
END_REGION

REGION Network 34: RO-01 ORP PROCESS VALVE ABV-302 OPEN COMMOND FAIL
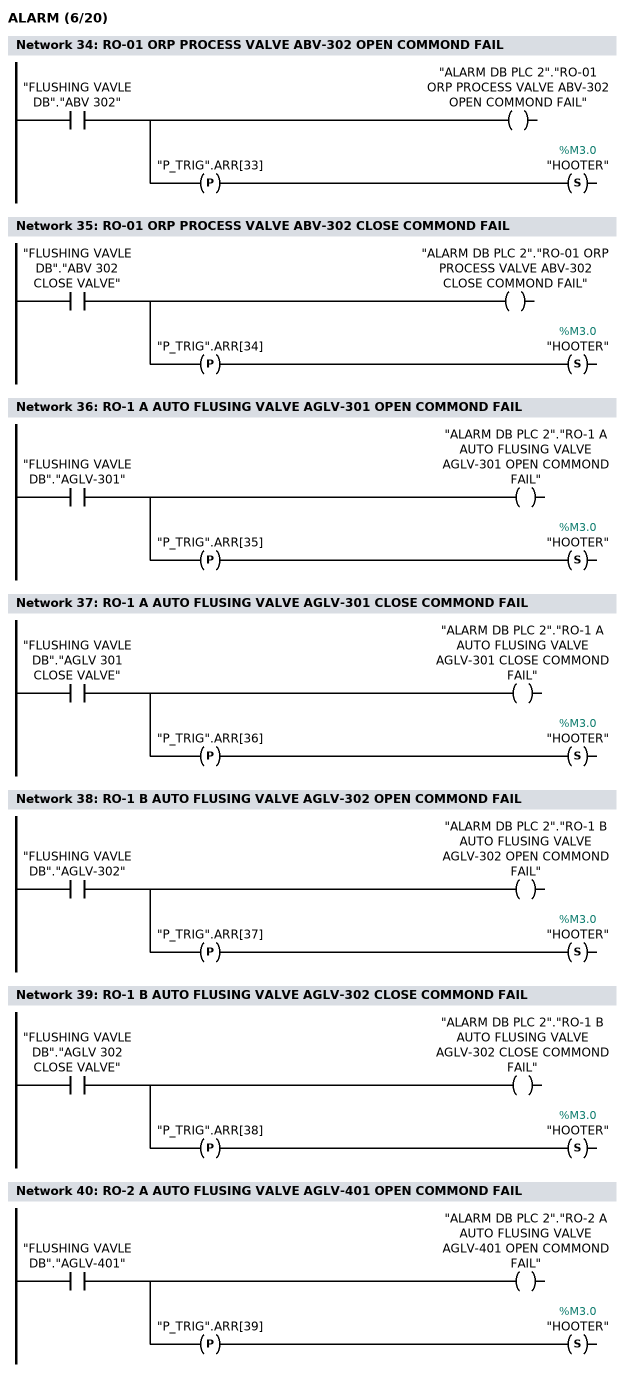
   RUNG wire#powerrail
      Contact( "FLUSHING VAVLE DB"."ABV 302" )
      wire#w1
      Coil( "ALARM DB PLC 2"."RO-01 ORP PROCESS VALVE ABV-302 OPEN COMMOND FAIL" )
   END_RUNG
   RUNG wire#w1
      P_Trig( "P_TRIG".ARR[33] )
      S_Coil( "HOOTER" )
   END_RUNG
   // the same network as SCL:
   "ALARM DB PLC 2"."RO-01 ORP PROCESS VALVE ABV-302 OPEN COMMOND FAIL" := "FLUSHING VAVLE DB"."ABV 302";
   #_w1 := "FLUSHING VAVLE DB"."ABV 302" AND NOT "P_TRIG".ARR[33];   // rising edge
   "P_TRIG".ARR[33] := "FLUSHING VAVLE DB"."ABV 302";
   IF #_w1 THEN "HOOTER" := TRUE; END_IF;
END_REGION

REGION Network 35: RO-01 ORP PROCESS VALVE ABV-302 CLOSE COMMOND FAIL
   RUNG wire#powerrail
      Contact( "FLUSHING VAVLE DB"."ABV 302 CLOSE VALVE" )
      wire#w1
      Coil( "ALARM DB PLC 2"."RO-01 ORP PROCESS VALVE ABV-302 CLOSE COMMOND FAIL" )
   END_RUNG
   RUNG wire#w1
      P_Trig( "P_TRIG".ARR[34] )
      S_Coil( "HOOTER" )
   END_RUNG
   // the same network as SCL:
   "ALARM DB PLC 2"."RO-01 ORP PROCESS VALVE ABV-302 CLOSE COMMOND FAIL" := "FLUSHING VAVLE DB"."ABV 302 CLOSE VALVE";
   #_w1 := "FLUSHING VAVLE DB"."ABV 302 CLOSE VALVE" AND NOT "P_TRIG".ARR[34];   // rising edge
   "P_TRIG".ARR[34] := "FLUSHING VAVLE DB"."ABV 302 CLOSE VALVE";
   IF #_w1 THEN "HOOTER" := TRUE; END_IF;
END_REGION

REGION Network 36: RO-1 A AUTO FLUSING VALVE AGLV-301 OPEN COMMOND FAIL
   RUNG wire#powerrail
      Contact( "FLUSHING VAVLE DB"."AGLV-301" )
      wire#w1
      Coil( "ALARM DB PLC 2"."RO-1 A AUTO FLUSING VALVE AGLV-301 OPEN COMMOND FAIL" )
   END_RUNG
   RUNG wire#w1
      P_Trig( "P_TRIG".ARR[35] )
      S_Coil( "HOOTER" )
   END_RUNG
   // the same network as SCL:
   "ALARM DB PLC 2"."RO-1 A AUTO FLUSING VALVE AGLV-301 OPEN COMMOND FAIL" := "FLUSHING VAVLE DB"."AGLV-301";
   #_w1 := "FLUSHING VAVLE DB"."AGLV-301" AND NOT "P_TRIG".ARR[35];   // rising edge
   "P_TRIG".ARR[35] := "FLUSHING VAVLE DB"."AGLV-301";
   IF #_w1 THEN "HOOTER" := TRUE; END_IF;
END_REGION

REGION Network 37: RO-1 A AUTO FLUSING VALVE AGLV-301 CLOSE COMMOND FAIL
   RUNG wire#powerrail
      Contact( "FLUSHING VAVLE DB"."AGLV 301 CLOSE VALVE" )
      wire#w1
      Coil( "ALARM DB PLC 2"."RO-1 A AUTO FLUSING VALVE AGLV-301 CLOSE COMMOND FAIL" )
   END_RUNG
   RUNG wire#w1
      P_Trig( "P_TRIG".ARR[36] )
      S_Coil( "HOOTER" )
   END_RUNG
   // the same network as SCL:
   "ALARM DB PLC 2"."RO-1 A AUTO FLUSING VALVE AGLV-301 CLOSE COMMOND FAIL" := "FLUSHING VAVLE DB"."AGLV 301 CLOSE VALVE";
   #_w1 := "FLUSHING VAVLE DB"."AGLV 301 CLOSE VALVE" AND NOT "P_TRIG".ARR[36];   // rising edge
   "P_TRIG".ARR[36] := "FLUSHING VAVLE DB"."AGLV 301 CLOSE VALVE";
   IF #_w1 THEN "HOOTER" := TRUE; END_IF;
END_REGION

REGION Network 38: RO-1 B AUTO FLUSING VALVE AGLV-302 OPEN COMMOND FAIL
   RUNG wire#powerrail
      Contact( "FLUSHING VAVLE DB"."AGLV-302" )
      wire#w1
      Coil( "ALARM DB PLC 2"."RO-1 B AUTO FLUSING VALVE AGLV-302 OPEN COMMOND FAIL" )
   END_RUNG
   RUNG wire#w1
      P_Trig( "P_TRIG".ARR[37] )
      S_Coil( "HOOTER" )
   END_RUNG
   // the same network as SCL:
   "ALARM DB PLC 2"."RO-1 B AUTO FLUSING VALVE AGLV-302 OPEN COMMOND FAIL" := "FLUSHING VAVLE DB"."AGLV-302";
   #_w1 := "FLUSHING VAVLE DB"."AGLV-302" AND NOT "P_TRIG".ARR[37];   // rising edge
   "P_TRIG".ARR[37] := "FLUSHING VAVLE DB"."AGLV-302";
   IF #_w1 THEN "HOOTER" := TRUE; END_IF;
END_REGION

REGION Network 39: RO-1 B AUTO FLUSING VALVE AGLV-302 CLOSE COMMOND FAIL
   RUNG wire#powerrail
      Contact( "FLUSHING VAVLE DB"."AGLV 302 CLOSE VALVE" )
      wire#w1
      Coil( "ALARM DB PLC 2"."RO-1 B AUTO FLUSING VALVE AGLV-302 CLOSE COMMOND FAIL" )
   END_RUNG
   RUNG wire#w1
      P_Trig( "P_TRIG".ARR[38] )
      S_Coil( "HOOTER" )
   END_RUNG
   // the same network as SCL:
   "ALARM DB PLC 2"."RO-1 B AUTO FLUSING VALVE AGLV-302 CLOSE COMMOND FAIL" := "FLUSHING VAVLE DB"."AGLV 302 CLOSE VALVE";
   #_w1 := "FLUSHING VAVLE DB"."AGLV 302 CLOSE VALVE" AND NOT "P_TRIG".ARR[38];   // rising edge
   "P_TRIG".ARR[38] := "FLUSHING VAVLE DB"."AGLV 302 CLOSE VALVE";
   IF #_w1 THEN "HOOTER" := TRUE; END_IF;
END_REGION

REGION Network 40: RO-2 A AUTO FLUSING VALVE AGLV-401 OPEN COMMOND FAIL
   RUNG wire#powerrail
      Contact( "FLUSHING VAVLE DB"."AGLV-401" )
      wire#w1
      Coil( "ALARM DB PLC 2"."RO-2 A AUTO FLUSING VALVE AGLV-401 OPEN COMMOND FAIL" )
   END_RUNG
   RUNG wire#w1
      P_Trig( "P_TRIG".ARR[39] )
      S_Coil( "HOOTER" )
   END_RUNG
   // the same network as SCL:
   "ALARM DB PLC 2"."RO-2 A AUTO FLUSING VALVE AGLV-401 OPEN COMMOND FAIL" := "FLUSHING VAVLE DB"."AGLV-401";
   #_w1 := "FLUSHING VAVLE DB"."AGLV-401" AND NOT "P_TRIG".ARR[39];   // rising edge
   "P_TRIG".ARR[39] := "FLUSHING VAVLE DB"."AGLV-401";
   IF #_w1 THEN "HOOTER" := TRUE; END_IF;
END_REGION

